REGION Network 2: 上行制动
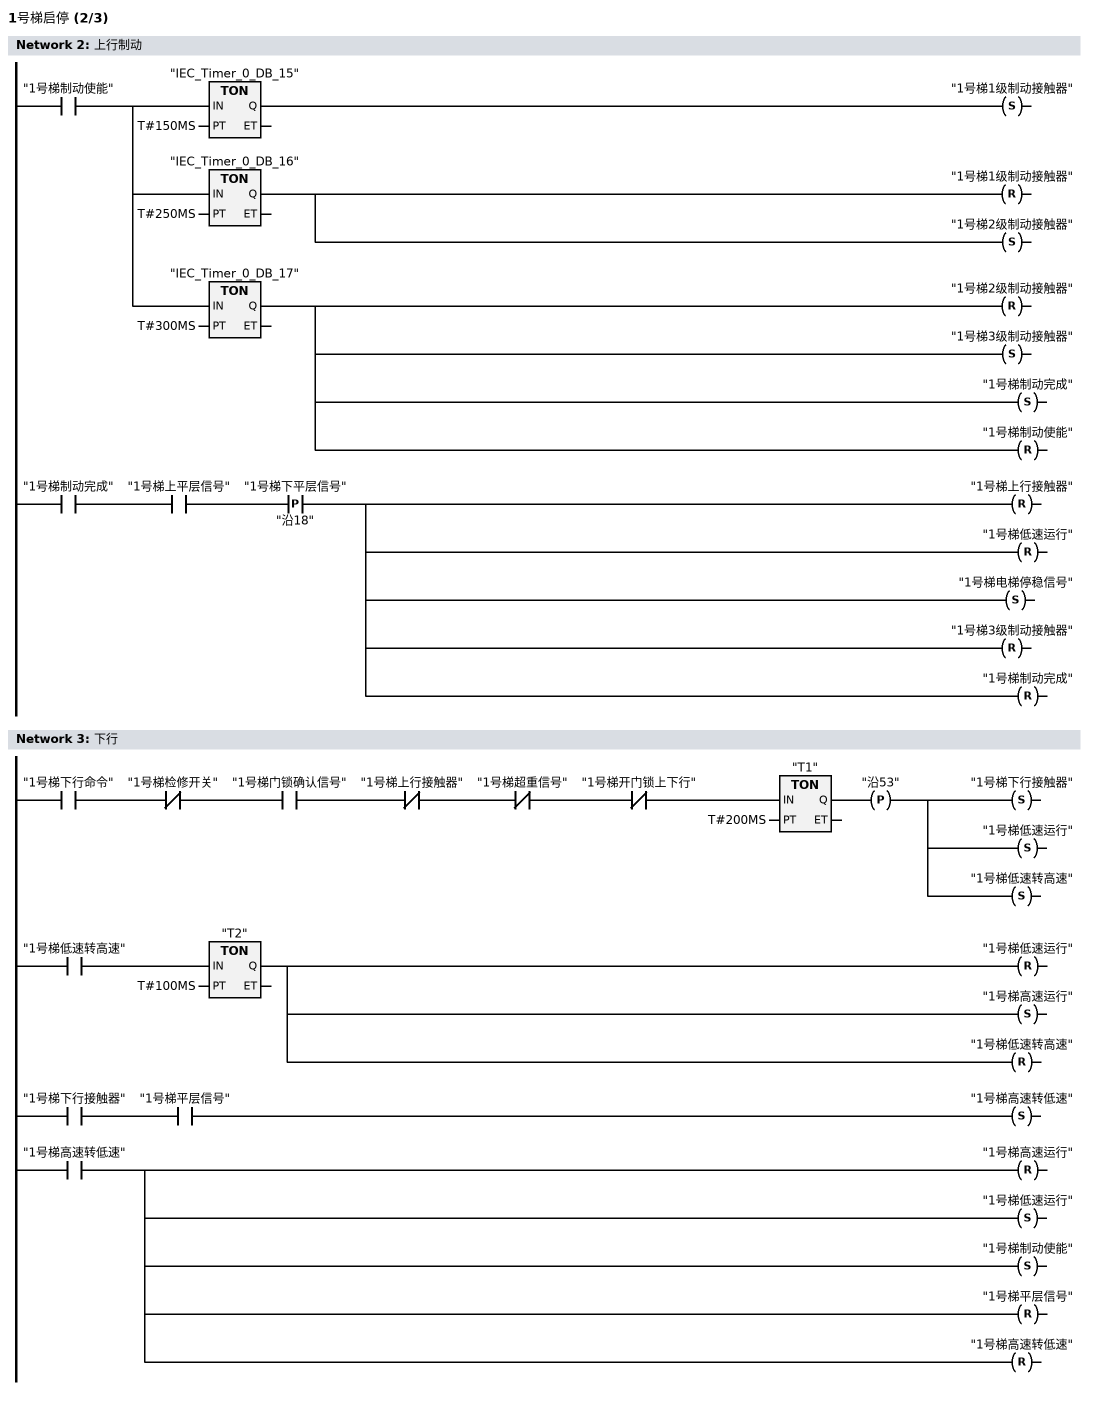
   "IEC_Timer_0_DB_15".TON(IN := "1号梯制动使能", PT := T#150MS);
   IF "IEC_Timer_0_DB_15".Q THEN "1号梯1级制动接触器" := TRUE; END_IF;
   "IEC_Timer_0_DB_16".TON(IN := "1号梯制动使能", PT := T#250MS);
   IF "IEC_Timer_0_DB_16".Q THEN
       "1号梯1级制动接触器" := FALSE;
       "1号梯2级制动接触器" := TRUE;
   END_IF;
   "IEC_Timer_0_DB_17".TON(IN := "1号梯制动使能", PT := T#300MS);
   IF "IEC_Timer_0_DB_17".Q THEN
       "1号梯2级制动接触器" := FALSE;
       "1号梯3级制动接触器" := TRUE;
       "1号梯制动完成" := TRUE;
       "1号梯制动使能" := FALSE;
   END_IF;
   #_w1 := "1号梯制动完成" AND "1号梯上平层信号" AND "1号梯下平层信号" AND NOT "沿18";   // rising edge of "1号梯下平层信号"
   "沿18" := "1号梯下平层信号";
   IF #_w1 THEN
       "1号梯上行接触器" := FALSE;
       "1号梯低速运行" := FALSE;
       "1号梯电梯停稳信号" := TRUE;
       "1号梯3级制动接触器" := FALSE;
       "1号梯制动完成" := FALSE;
   END_IF;
END_REGION

REGION Network 3: 下行
   "T1".TON(IN := "1号梯下行命令" AND NOT "1号梯检修开关" AND "1号梯门锁确认信号" AND NOT "1号梯上行接触器" AND NOT "1号梯超重信号" AND NOT "1号梯开门锁上下行",
            PT := T#200MS);
   #_w1 := "T1".Q AND NOT "沿53";   // rising edge
   "沿53" := "T1".Q;
   IF #_w1 THEN
       "1号梯下行接触器" := TRUE;
       "1号梯低速运行" := TRUE;
       "1号梯低速转高速" := TRUE;
   END_IF;
   "T2".TON(IN := "1号梯低速转高速", PT := T#100MS);
   IF "T2".Q THEN
       "1号梯低速运行" := FALSE;
       "1号梯高速运行" := TRUE;
       "1号梯低速转高速" := FALSE;
   END_IF;
   IF "1号梯下行接触器" AND "1号梯平层信号" THEN "1号梯高速转低速" := TRUE; END_IF;
   IF "1号梯高速转低速" THEN
       "1号梯高速运行" := FALSE;
       "1号梯低速运行" := TRUE;
       "1号梯制动使能" := TRUE;
       "1号梯平层信号" := FALSE;
       "1号梯高速转低速" := FALSE;
   END_IF;
END_REGION

REGION Network 4: 下行制动
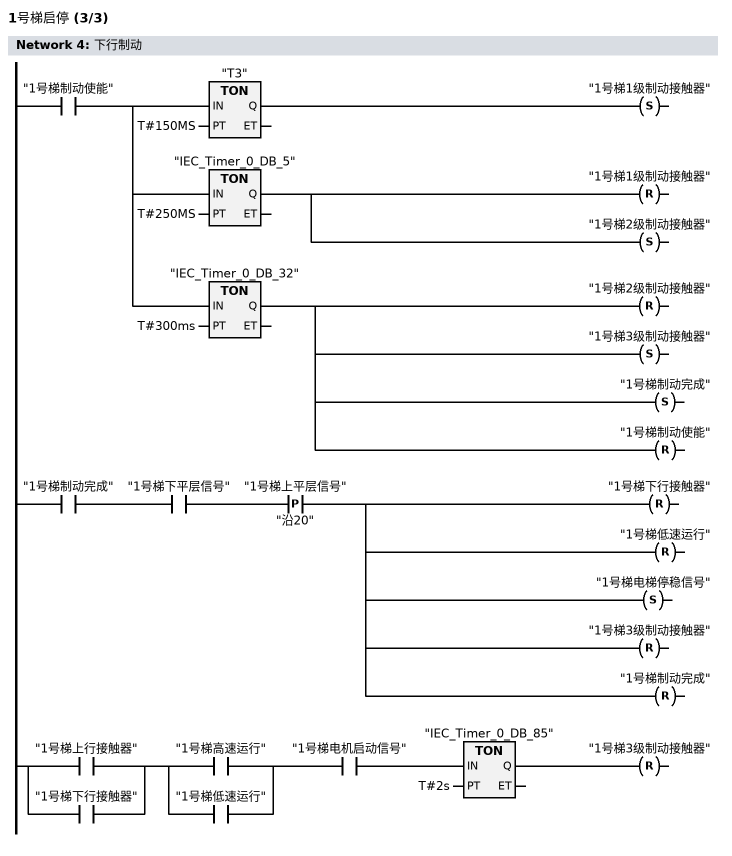
   "T3".TON(IN := "1号梯制动使能", PT := T#150MS);
   IF "T3".Q THEN "1号梯1级制动接触器" := TRUE; END_IF;
   "IEC_Timer_0_DB_5".TON(IN := "1号梯制动使能", PT := T#250MS);
   IF "IEC_Timer_0_DB_5".Q THEN
       "1号梯1级制动接触器" := FALSE;
       "1号梯2级制动接触器" := TRUE;
   END_IF;
   "IEC_Timer_0_DB_32".TON(IN := "1号梯制动使能", PT := T#300ms);
   IF "IEC_Timer_0_DB_32".Q THEN
       "1号梯2级制动接触器" := FALSE;
       "1号梯3级制动接触器" := TRUE;
       "1号梯制动完成" := TRUE;
       "1号梯制动使能" := FALSE;
   END_IF;
   #_w1 := "1号梯制动完成" AND "1号梯下平层信号" AND "1号梯上平层信号" AND NOT "沿20";   // rising edge of "1号梯上平层信号"
   "沿20" := "1号梯上平层信号";
   IF #_w1 THEN
       "1号梯下行接触器" := FALSE;
       "1号梯低速运行" := FALSE;
       "1号梯电梯停稳信号" := TRUE;
       "1号梯3级制动接触器" := FALSE;
       "1号梯制动完成" := FALSE;
   END_IF;
   "IEC_Timer_0_DB_85".TON(IN := ("1号梯上行接触器" OR "1号梯下行接触器") AND ("1号梯高速运行" OR "1号梯低速运行") AND "1号梯电机启动信号",
                           PT := T#2s);
   IF "IEC_Timer_0_DB_85".Q THEN "1号梯3级制动接触器" := FALSE; END_IF;
END_REGION
END_FUNCTION

FUNCTION "1号梯顺向截梯" : Void   // FC18, LAD
{ S7_Optimized_Access := 'TRUE' }
VERSION : 0.1
BEGIN

REGION Network 1: 上行拦截电梯
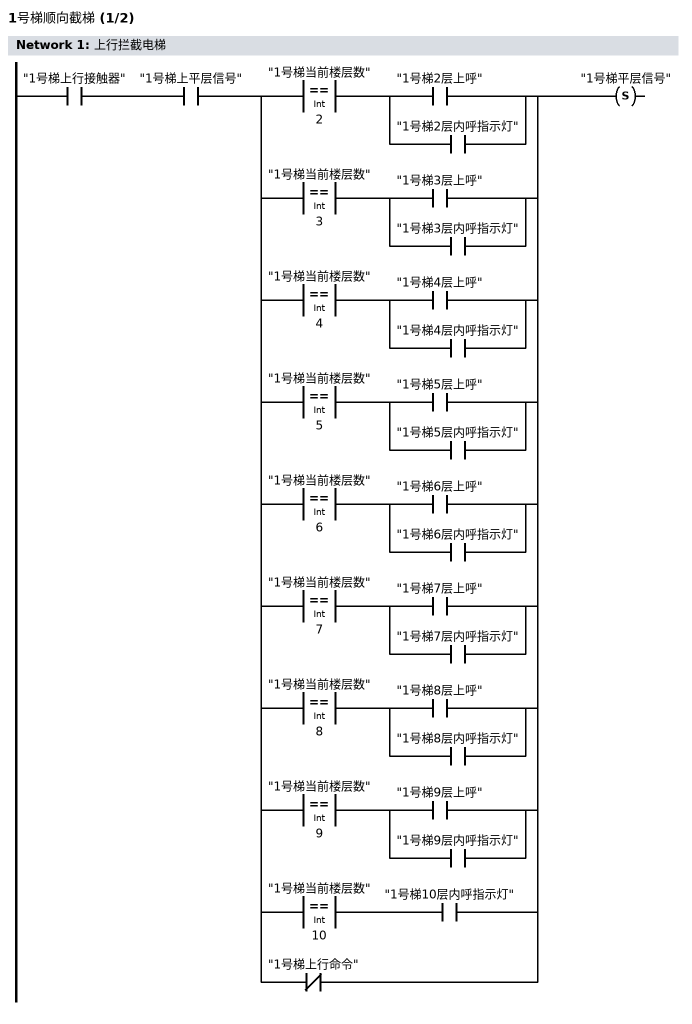
   RUNG wire#powerrail
      Contact( "1号梯上行接触器" )
      Contact( "1号梯上平层信号" )
      wire#w1
      { S7_Templates := "SrcType := Int" } EQ_Contact(in1 := "1号梯当前楼层数", in2 := 2)
      wire#w2
      Contact( "1号梯2层上呼" )
      wire#w3
      S_Coil( "1号梯平层信号" )
   END_RUNG
   RUNG wire#w2
      Contact( "1号梯2层内呼指示灯" )
   END_RUNG wire#w3
   RUNG wire#w1
      { S7_Templates := "SrcType := Int" } EQ_Contact(in1 := "1号梯当前楼层数", in2 := 3)
      wire#w4
      Contact( "1号梯3层上呼" )
   END_RUNG wire#w3
   RUNG wire#w4
      Contact( "1号梯3层内呼指示灯" )
   END_RUNG wire#w3
   RUNG wire#w1
      { S7_Templates := "SrcType := Int" } EQ_Contact(in1 := "1号梯当前楼层数", in2 := 4)
      wire#w5
      Contact( "1号梯4层上呼" )
   END_RUNG wire#w3
   RUNG wire#w5
      Contact( "1号梯4层内呼指示灯" )
   END_RUNG wire#w3
   RUNG wire#w1
      { S7_Templates := "SrcType := Int" } EQ_Contact(in1 := "1号梯当前楼层数", in2 := 5)
      wire#w6
      Contact( "1号梯5层上呼" )
   END_RUNG wire#w3
   RUNG wire#w6
      Contact( "1号梯5层内呼指示灯" )
   END_RUNG wire#w3
   RUNG wire#w1
      { S7_Templates := "SrcType := Int" } EQ_Contact(in1 := "1号梯当前楼层数", in2 := 6)
      wire#w7
      Contact( "1号梯6层上呼" )
   END_RUNG wire#w3
   RUNG wire#w7
      Contact( "1号梯6层内呼指示灯" )
   END_RUNG wire#w3
   RUNG wire#w1
      { S7_Templates := "SrcType := Int" } EQ_Contact(in1 := "1号梯当前楼层数", in2 := 7)
      wire#w8
      Contact( "1号梯7层上呼" )
   END_RUNG wire#w3
   RUNG wire#w8
      Contact( "1号梯7层内呼指示灯" )
   END_RUNG wire#w3
   RUNG wire#w1
      { S7_Templates := "SrcType := Int" } EQ_Contact(in1 := "1号梯当前楼层数", in2 := 8)
      wire#w9
      Contact( "1号梯8层上呼" )
   END_RUNG wire#w3
   RUNG wire#w9
      Contact( "1号梯8层内呼指示灯" )
   END_RUNG wire#w3
   RUNG wire#w1
      { S7_Templates := "SrcType := Int" } EQ_Contact(in1 := "1号梯当前楼层数", in2 := 9)
      wire#w10
      Contact( "1号梯9层上呼" )
   END_RUNG wire#w3
   RUNG wire#w10
      Contact( "1号梯9层内呼指示灯" )
   END_RUNG wire#w3
   RUNG wire#w1
      { S7_Templates := "SrcType := Int" } EQ_Contact(in1 := "1号梯当前楼层数", in2 := 10)
      Contact( "1号梯10层内呼指示灯" )
   END_RUNG wire#w3
   RUNG wire#w1
      I_Contact( "1号梯上行命令" )
   END_RUNG wire#w3
   // the same network as SCL:
   IF "1号梯上行接触器" AND "1号梯上平层信号" AND ((("1号梯当前楼层数" = 2) AND ("1号梯2层上呼" OR "1号梯2层内呼指示灯")) OR (("1号梯当前楼层数" = 3) AND ("1号梯3层上呼" OR "1号梯3层内呼指示灯")) OR (("1号梯当前楼层数" = 4) AND ("1号梯4层上呼" OR "1号梯4层内呼指示灯")) OR (("1号梯当前楼层数" = 5) AND ("1号梯5层上呼" OR "1号梯5层内呼指示灯")) OR (("1号梯当前楼层数" = 6) AND ("1号梯6层上呼" OR "1号梯6层内呼指示灯")) OR (("1号梯当前楼层数" = 7) AND ("1号梯7层上呼" OR "1号梯7层内呼指示灯")) OR (("1号梯当前楼层数" = 8) AND ("1号梯8层上呼" OR "1号梯8层内呼指示灯")) OR (("1号梯当前楼层数" = 9) AND ("1号梯9层上呼" OR "1号梯9层内呼指示灯")) OR (("1号梯当前楼层数" = 10) AND "1号梯10层内呼指示灯") OR NOT "1号梯上行命令") THEN
       "1号梯平层信号" := TRUE;
   END_IF;
END_REGION

REGION Network 2: 下行拦截电梯
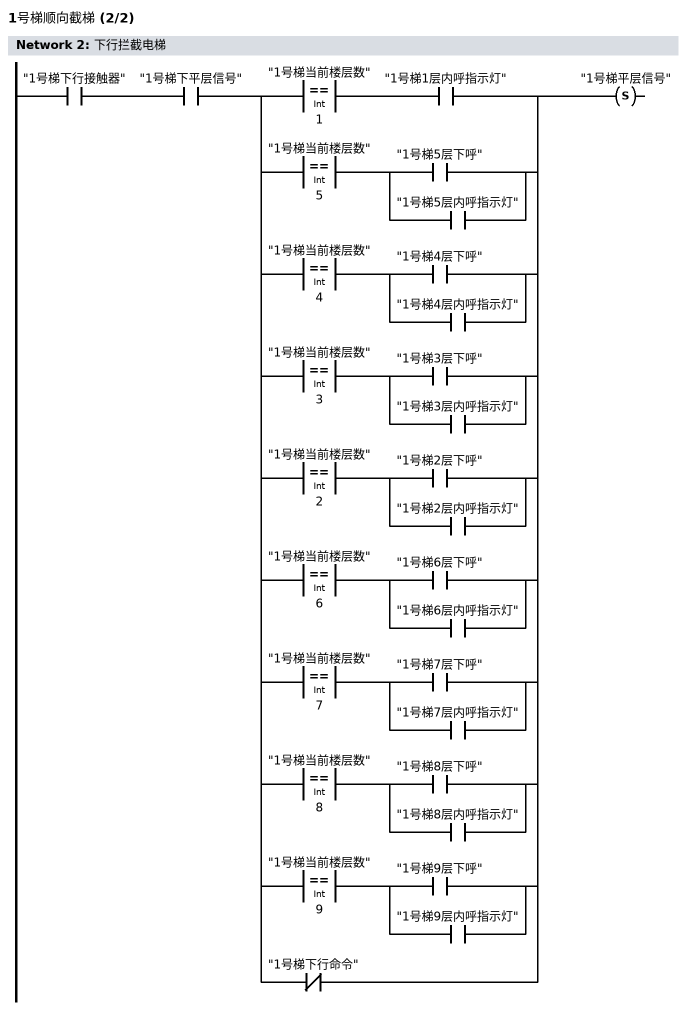
   RUNG wire#powerrail
      Contact( "1号梯下行接触器" )
      Contact( "1号梯下平层信号" )
      wire#w1
      { S7_Templates := "SrcType := Int" } EQ_Contact(in1 := "1号梯当前楼层数", in2 := 1)
      Contact( "1号梯1层内呼指示灯" )
      wire#w2
      S_Coil( "1号梯平层信号" )
   END_RUNG
   RUNG wire#w1
      { S7_Templates := "SrcType := Int" } EQ_Contact(in1 := "1号梯当前楼层数", in2 := 5)
      wire#w3
      Contact( "1号梯5层下呼" )
   END_RUNG wire#w2
   RUNG wire#w3
      Contact( "1号梯5层内呼指示灯" )
   END_RUNG wire#w2
   RUNG wire#w1
      { S7_Templates := "SrcType := Int" } EQ_Contact(in1 := "1号梯当前楼层数", in2 := 4)
      wire#w4
      Contact( "1号梯4层下呼" )
   END_RUNG wire#w2
   RUNG wire#w4
      Contact( "1号梯4层内呼指示灯" )
   END_RUNG wire#w2
   RUNG wire#w1
      { S7_Templates := "SrcType := Int" } EQ_Contact(in1 := "1号梯当前楼层数", in2 := 3)
      wire#w5
      Contact( "1号梯3层下呼" )
   END_RUNG wire#w2
   RUNG wire#w5
      Contact( "1号梯3层内呼指示灯" )
   END_RUNG wire#w2
   RUNG wire#w1
      { S7_Templates := "SrcType := Int" } EQ_Contact(in1 := "1号梯当前楼层数", in2 := 2)
      wire#w6
      Contact( "1号梯2层下呼" )
   END_RUNG wire#w2
   RUNG wire#w6
      Contact( "1号梯2层内呼指示灯" )
   END_RUNG wire#w2
   RUNG wire#w1
      { S7_Templates := "SrcType := Int" } EQ_Contact(in1 := "1号梯当前楼层数", in2 := 6)
      wire#w7
      Contact( "1号梯6层下呼" )
   END_RUNG wire#w2
   RUNG wire#w7
      Contact( "1号梯6层内呼指示灯" )
   END_RUNG wire#w2
   RUNG wire#w1
      { S7_Templates := "SrcType := Int" } EQ_Contact(in1 := "1号梯当前楼层数", in2 := 7)
      wire#w8
      Contact( "1号梯7层下呼" )
   END_RUNG wire#w2
   RUNG wire#w8
      Contact( "1号梯7层内呼指示灯" )
   END_RUNG wire#w2
   RUNG wire#w1
      { S7_Templates := "SrcType := Int" } EQ_Contact(in1 := "1号梯当前楼层数", in2 := 8)
      wire#w9
      Contact( "1号梯8层下呼" )
   END_RUNG wire#w2
   RUNG wire#w9
      Contact( "1号梯8层内呼指示灯" )
   END_RUNG wire#w2
   RUNG wire#w1
      { S7_Templates := "SrcType := Int" } EQ_Contact(in1 := "1号梯当前楼层数", in2 := 9)
      wire#w10
      Contact( "1号梯9层下呼" )
   END_RUNG wire#w2
   RUNG wire#w10
      Contact( "1号梯9层内呼指示灯" )
   END_RUNG wire#w2
   RUNG wire#w1
      I_Contact( "1号梯下行命令" )
   END_RUNG wire#w2
   // the same network as SCL:
   IF "1号梯下行接触器" AND "1号梯下平层信号" AND ((("1号梯当前楼层数" = 1) AND "1号梯1层内呼指示灯") OR (("1号梯当前楼层数" = 5) AND ("1号梯5层下呼" OR "1号梯5层内呼指示灯")) OR (("1号梯当前楼层数" = 4) AND ("1号梯4层下呼" OR "1号梯4层内呼指示灯")) OR (("1号梯当前楼层数" = 3) AND ("1号梯3层下呼" OR "1号梯3层内呼指示灯")) OR (("1号梯当前楼层数" = 2) AND ("1号梯2层下呼" OR "1号梯2层内呼指示灯")) OR (("1号梯当前楼层数" = 6) AND ("1号梯6层下呼" OR "1号梯6层内呼指示灯")) OR (("1号梯当前楼层数" = 7) AND ("1号梯7层下呼" OR "1号梯7层内呼指示灯")) OR (("1号梯当前楼层数" = 8) AND ("1号梯8层下呼" OR "1号梯8层内呼指示灯")) OR (("1号梯当前楼层数" = 9) AND ("1号梯9层下呼" OR "1号梯9层内呼指示灯")) OR NOT "1号梯下行命令") THEN
       "1号梯平层信号" := TRUE;
   END_IF;
END_REGION
END_FUNCTION

FUNCTION "1号梯轿内指示灯控制" : Void   // FC19, LAD
{ S7_Optimized_Access := 'TRUE' }
VERSION : 0.1
   VAR_TEMP   // added for the SCL form of the ladder/FBD networks
      _w1 : Bool;
      _w2 : Bool;
   END_VAR
BEGIN

REGION Network 1: 平层灭灯
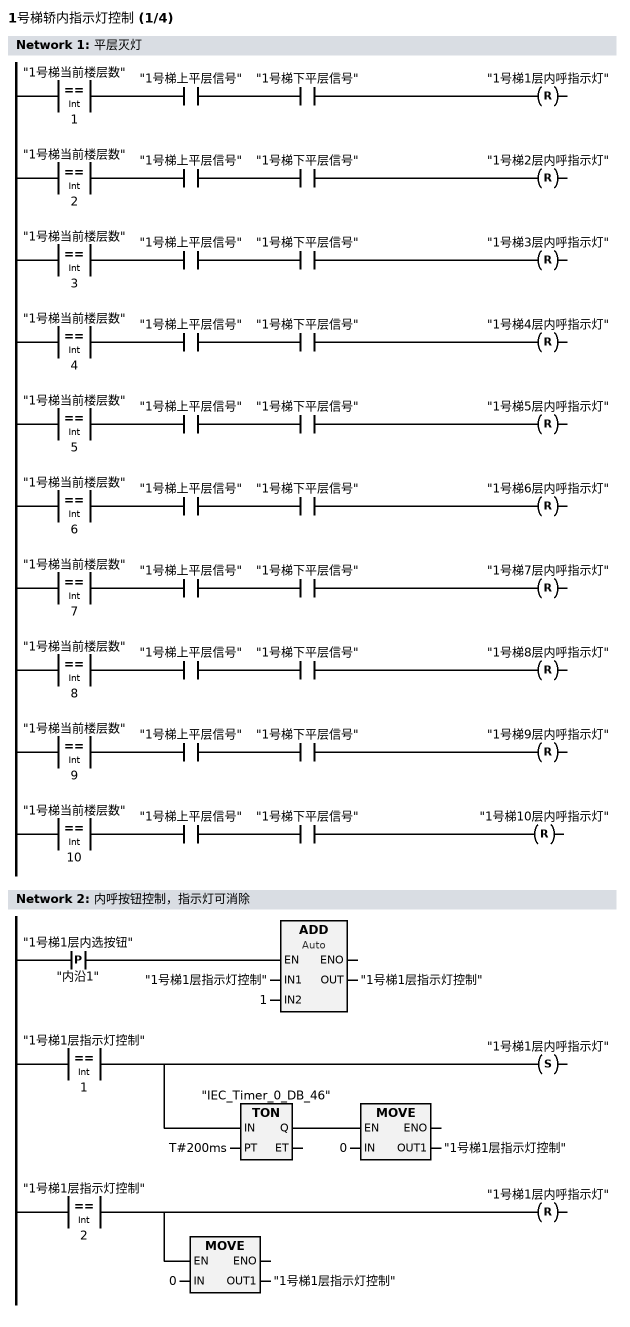
   RUNG wire#powerrail
      { S7_Templates := "SrcType := Int" } EQ_Contact(in1 := "1号梯当前楼层数", in2 := 1)
      Contact( "1号梯上平层信号" )
      Contact( "1号梯下平层信号" )
      R_Coil( "1号梯1层内呼指示灯" )
   END_RUNG
   RUNG wire#powerrail
      { S7_Templates := "SrcType := Int" } EQ_Contact(in1 := "1号梯当前楼层数", in2 := 2)
      Contact( "1号梯上平层信号" )
      Contact( "1号梯下平层信号" )
      R_Coil( "1号梯2层内呼指示灯" )
   END_RUNG
   RUNG wire#powerrail
      { S7_Templates := "SrcType := Int" } EQ_Contact(in1 := "1号梯当前楼层数", in2 := 3)
      Contact( "1号梯上平层信号" )
      Contact( "1号梯下平层信号" )
      R_Coil( "1号梯3层内呼指示灯" )
   END_RUNG
   RUNG wire#powerrail
      { S7_Templates := "SrcType := Int" } EQ_Contact(in1 := "1号梯当前楼层数", in2 := 4)
      Contact( "1号梯上平层信号" )
      Contact( "1号梯下平层信号" )
      R_Coil( "1号梯4层内呼指示灯" )
   END_RUNG
   RUNG wire#powerrail
      { S7_Templates := "SrcType := Int" } EQ_Contact(in1 := "1号梯当前楼层数", in2 := 5)
      Contact( "1号梯上平层信号" )
      Contact( "1号梯下平层信号" )
      R_Coil( "1号梯5层内呼指示灯" )
   END_RUNG
   RUNG wire#powerrail
      { S7_Templates := "SrcType := Int" } EQ_Contact(in1 := "1号梯当前楼层数", in2 := 6)
      Contact( "1号梯上平层信号" )
      Contact( "1号梯下平层信号" )
      R_Coil( "1号梯6层内呼指示灯" )
   END_RUNG
   RUNG wire#powerrail
      { S7_Templates := "SrcType := Int" } EQ_Contact(in1 := "1号梯当前楼层数", in2 := 7)
      Contact( "1号梯上平层信号" )
      Contact( "1号梯下平层信号" )
      R_Coil( "1号梯7层内呼指示灯" )
   END_RUNG
   RUNG wire#powerrail
      { S7_Templates := "SrcType := Int" } EQ_Contact(in1 := "1号梯当前楼层数", in2 := 8)
      Contact( "1号梯上平层信号" )
      Contact( "1号梯下平层信号" )
      R_Coil( "1号梯8层内呼指示灯" )
   END_RUNG
   RUNG wire#powerrail
      { S7_Templates := "SrcType := Int" } EQ_Contact(in1 := "1号梯当前楼层数", in2 := 9)
      Contact( "1号梯上平层信号" )
      Contact( "1号梯下平层信号" )
      R_Coil( "1号梯9层内呼指示灯" )
   END_RUNG
   RUNG wire#powerrail
      { S7_Templates := "SrcType := Int" } EQ_Contact(in1 := "1号梯当前楼层数", in2 := 10)
      Contact( "1号梯上平层信号" )
      Contact( "1号梯下平层信号" )
      R_Coil( "1号梯10层内呼指示灯" )
   END_RUNG
   // the same network as SCL:
   IF ("1号梯当前楼层数" = 1) AND "1号梯上平层信号" AND "1号梯下平层信号" THEN "1号梯1层内呼指示灯" := FALSE; END_IF;
   IF ("1号梯当前楼层数" = 2) AND "1号梯上平层信号" AND "1号梯下平层信号" THEN "1号梯2层内呼指示灯" := FALSE; END_IF;
   IF ("1号梯当前楼层数" = 3) AND "1号梯上平层信号" AND "1号梯下平层信号" THEN "1号梯3层内呼指示灯" := FALSE; END_IF;
   IF ("1号梯当前楼层数" = 4) AND "1号梯上平层信号" AND "1号梯下平层信号" THEN "1号梯4层内呼指示灯" := FALSE; END_IF;
   IF ("1号梯当前楼层数" = 5) AND "1号梯上平层信号" AND "1号梯下平层信号" THEN "1号梯5层内呼指示灯" := FALSE; END_IF;
   IF ("1号梯当前楼层数" = 6) AND "1号梯上平层信号" AND "1号梯下平层信号" THEN "1号梯6层内呼指示灯" := FALSE; END_IF;
   IF ("1号梯当前楼层数" = 7) AND "1号梯上平层信号" AND "1号梯下平层信号" THEN "1号梯7层内呼指示灯" := FALSE; END_IF;
   IF ("1号梯当前楼层数" = 8) AND "1号梯上平层信号" AND "1号梯下平层信号" THEN "1号梯8层内呼指示灯" := FALSE; END_IF;
   IF ("1号梯当前楼层数" = 9) AND "1号梯上平层信号" AND "1号梯下平层信号" THEN "1号梯9层内呼指示灯" := FALSE; END_IF;
   IF ("1号梯当前楼层数" = 10) AND "1号梯上平层信号" AND "1号梯下平层信号" THEN "1号梯10层内呼指示灯" := FALSE; END_IF;
END_REGION

REGION Network 2: 内呼按钮控制，指示灯可消除
   #_w1 := "1号梯1层内选按钮" AND NOT "内沿1";   // rising edge of "1号梯1层内选按钮"
   "内沿1" := "1号梯1层内选按钮";
   IF #_w1 THEN "1号梯1层指示灯控制" := "1号梯1层指示灯控制" + 1; END_IF;
   #_w2 := "1号梯1层指示灯控制" = 1;
   IF #_w2 THEN "1号梯1层内呼指示灯" := TRUE; END_IF;
   "IEC_Timer_0_DB_46".TON(IN := #_w2, PT := T#200ms);
   IF "IEC_Timer_0_DB_46".Q THEN "1号梯1层指示灯控制" := 0; END_IF;
   IF "1号梯1层指示灯控制" = 2 THEN
       "1号梯1层内呼指示灯" := FALSE;
       "1号梯1层指示灯控制" := 0;
   END_IF;
END_REGION

REGION Network 3: 内呼按钮控制，指示灯可消除
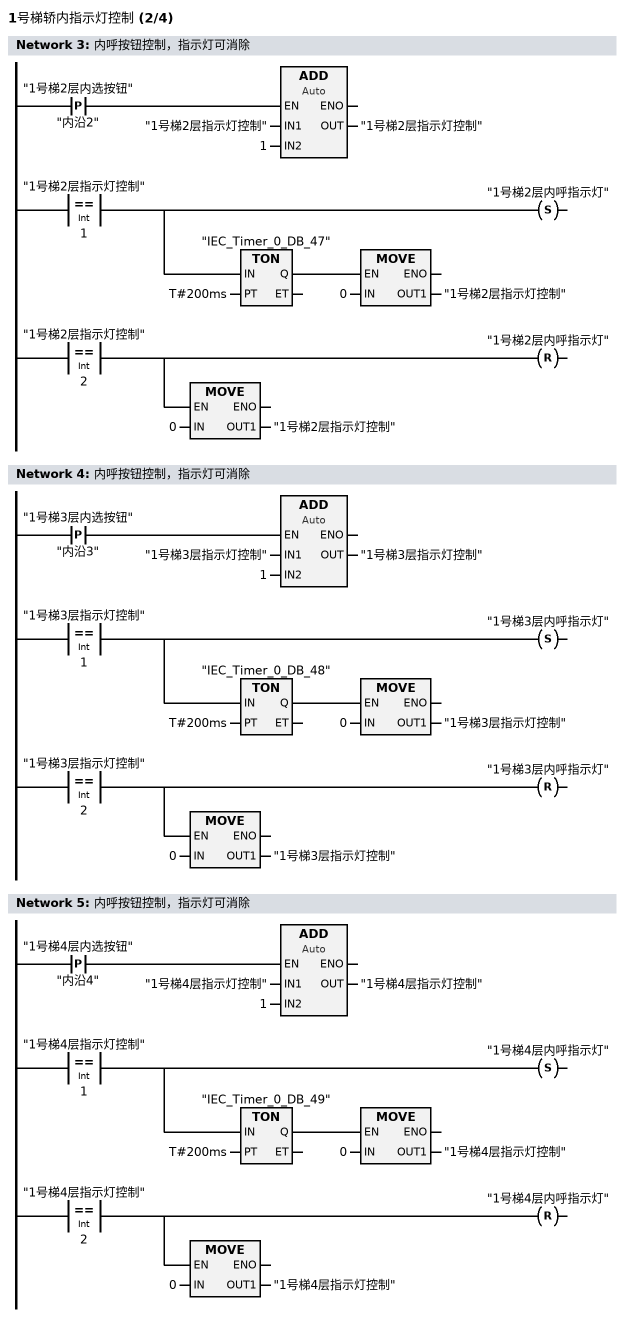
   #_w1 := "1号梯2层内选按钮" AND NOT "内沿2";   // rising edge of "1号梯2层内选按钮"
   "内沿2" := "1号梯2层内选按钮";
   IF #_w1 THEN "1号梯2层指示灯控制" := "1号梯2层指示灯控制" + 1; END_IF;
   #_w2 := "1号梯2层指示灯控制" = 1;
   IF #_w2 THEN "1号梯2层内呼指示灯" := TRUE; END_IF;
   "IEC_Timer_0_DB_47".TON(IN := #_w2, PT := T#200ms);
   IF "IEC_Timer_0_DB_47".Q THEN "1号梯2层指示灯控制" := 0; END_IF;
   IF "1号梯2层指示灯控制" = 2 THEN
       "1号梯2层内呼指示灯" := FALSE;
       "1号梯2层指示灯控制" := 0;
   END_IF;
END_REGION

REGION Network 4: 内呼按钮控制，指示灯可消除
   #_w1 := "1号梯3层内选按钮" AND NOT "内沿3";   // rising edge of "1号梯3层内选按钮"
   "内沿3" := "1号梯3层内选按钮";
   IF #_w1 THEN "1号梯3层指示灯控制" := "1号梯3层指示灯控制" + 1; END_IF;
   #_w2 := "1号梯3层指示灯控制" = 1;
   IF #_w2 THEN "1号梯3层内呼指示灯" := TRUE; END_IF;
   "IEC_Timer_0_DB_48".TON(IN := #_w2, PT := T#200ms);
   IF "IEC_Timer_0_DB_48".Q THEN "1号梯3层指示灯控制" := 0; END_IF;
   IF "1号梯3层指示灯控制" = 2 THEN
       "1号梯3层内呼指示灯" := FALSE;
       "1号梯3层指示灯控制" := 0;
   END_IF;
END_REGION

REGION Network 5: 内呼按钮控制，指示灯可消除
   #_w1 := "1号梯4层内选按钮" AND NOT "内沿4";   // rising edge of "1号梯4层内选按钮"
   "内沿4" := "1号梯4层内选按钮";
   IF #_w1 THEN "1号梯4层指示灯控制" := "1号梯4层指示灯控制" + 1; END_IF;
   #_w2 := "1号梯4层指示灯控制" = 1;
   IF #_w2 THEN "1号梯4层内呼指示灯" := TRUE; END_IF;
   "IEC_Timer_0_DB_49".TON(IN := #_w2, PT := T#200ms);
   IF "IEC_Timer_0_DB_49".Q THEN "1号梯4层指示灯控制" := 0; END_IF;
   IF "1号梯4层指示灯控制" = 2 THEN
       "1号梯4层内呼指示灯" := FALSE;
       "1号梯4层指示灯控制" := 0;
   END_IF;
END_REGION

REGION Network 6: 内呼按钮控制，指示灯可消除
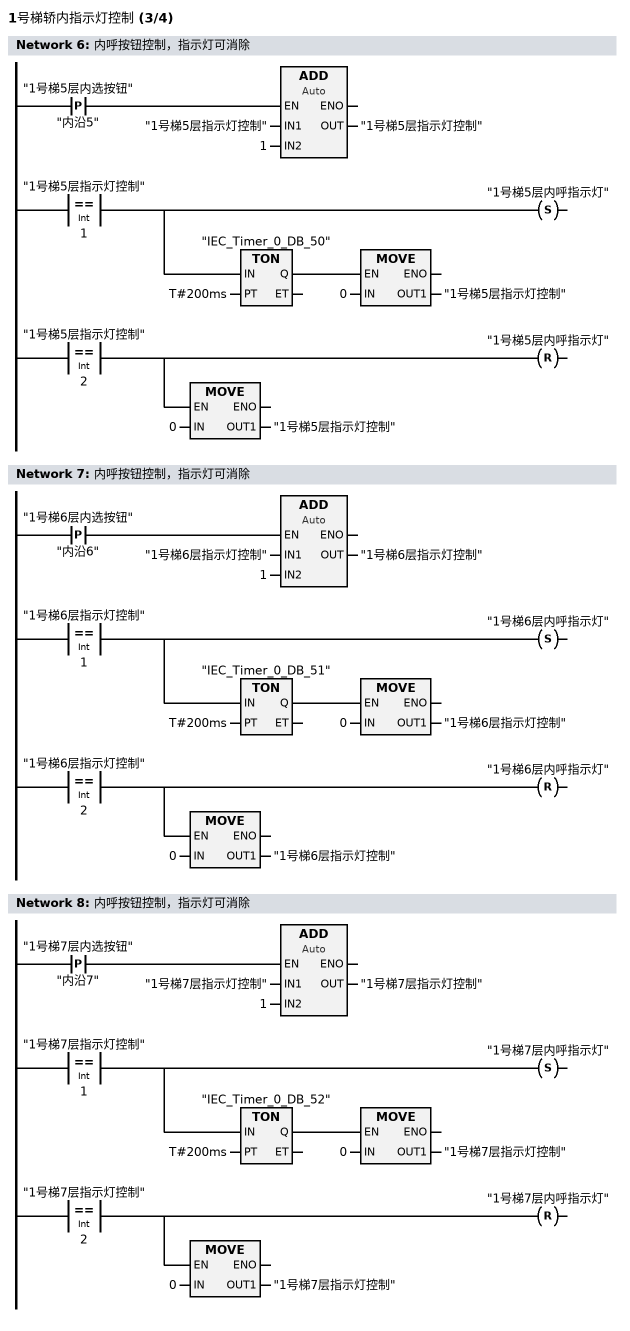
   #_w1 := "1号梯5层内选按钮" AND NOT "内沿5";   // rising edge of "1号梯5层内选按钮"
   "内沿5" := "1号梯5层内选按钮";
   IF #_w1 THEN "1号梯5层指示灯控制" := "1号梯5层指示灯控制" + 1; END_IF;
   #_w2 := "1号梯5层指示灯控制" = 1;
   IF #_w2 THEN "1号梯5层内呼指示灯" := TRUE; END_IF;
   "IEC_Timer_0_DB_50".TON(IN := #_w2, PT := T#200ms);
   IF "IEC_Timer_0_DB_50".Q THEN "1号梯5层指示灯控制" := 0; END_IF;
   IF "1号梯5层指示灯控制" = 2 THEN
       "1号梯5层内呼指示灯" := FALSE;
       "1号梯5层指示灯控制" := 0;
   END_IF;
END_REGION

REGION Network 7: 内呼按钮控制，指示灯可消除
   #_w1 := "1号梯6层内选按钮" AND NOT "内沿6";   // rising edge of "1号梯6层内选按钮"
   "内沿6" := "1号梯6层内选按钮";
   IF #_w1 THEN "1号梯6层指示灯控制" := "1号梯6层指示灯控制" + 1; END_IF;
   #_w2 := "1号梯6层指示灯控制" = 1;
   IF #_w2 THEN "1号梯6层内呼指示灯" := TRUE; END_IF;
   "IEC_Timer_0_DB_51".TON(IN := #_w2, PT := T#200ms);
   IF "IEC_Timer_0_DB_51".Q THEN "1号梯6层指示灯控制" := 0; END_IF;
   IF "1号梯6层指示灯控制" = 2 THEN
       "1号梯6层内呼指示灯" := FALSE;
       "1号梯6层指示灯控制" := 0;
   END_IF;
END_REGION

REGION Network 8: 内呼按钮控制，指示灯可消除
   #_w1 := "1号梯7层内选按钮" AND NOT "内沿7";   // rising edge of "1号梯7层内选按钮"
   "内沿7" := "1号梯7层内选按钮";
   IF #_w1 THEN "1号梯7层指示灯控制" := "1号梯7层指示灯控制" + 1; END_IF;
   #_w2 := "1号梯7层指示灯控制" = 1;
   IF #_w2 THEN "1号梯7层内呼指示灯" := TRUE; END_IF;
   "IEC_Timer_0_DB_52".TON(IN := #_w2, PT := T#200ms);
   IF "IEC_Timer_0_DB_52".Q THEN "1号梯7层指示灯控制" := 0; END_IF;
   IF "1号梯7层指示灯控制" = 2 THEN
       "1号梯7层内呼指示灯" := FALSE;
       "1号梯7层指示灯控制" := 0;
   END_IF;
END_REGION

REGION Network 9: 内呼按钮控制，指示灯可消除
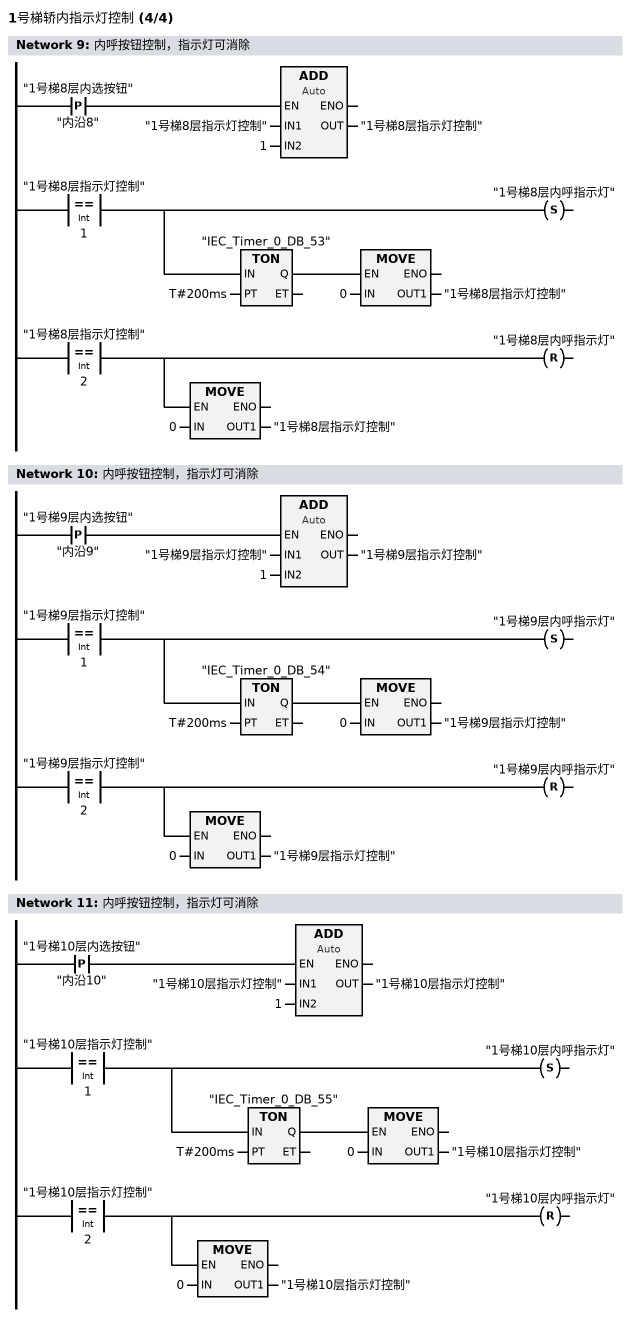
   #_w1 := "1号梯8层内选按钮" AND NOT "内沿8";   // rising edge of "1号梯8层内选按钮"
   "内沿8" := "1号梯8层内选按钮";
   IF #_w1 THEN "1号梯8层指示灯控制" := "1号梯8层指示灯控制" + 1; END_IF;
   #_w2 := "1号梯8层指示灯控制" = 1;
   IF #_w2 THEN "1号梯8层内呼指示灯" := TRUE; END_IF;
   "IEC_Timer_0_DB_53".TON(IN := #_w2, PT := T#200ms);
   IF "IEC_Timer_0_DB_53".Q THEN "1号梯8层指示灯控制" := 0; END_IF;
   IF "1号梯8层指示灯控制" = 2 THEN
       "1号梯8层内呼指示灯" := FALSE;
       "1号梯8层指示灯控制" := 0;
   END_IF;
END_REGION

REGION Network 10: 内呼按钮控制，指示灯可消除
   #_w1 := "1号梯9层内选按钮" AND NOT "内沿9";   // rising edge of "1号梯9层内选按钮"
   "内沿9" := "1号梯9层内选按钮";
   IF #_w1 THEN "1号梯9层指示灯控制" := "1号梯9层指示灯控制" + 1; END_IF;
   #_w2 := "1号梯9层指示灯控制" = 1;
   IF #_w2 THEN "1号梯9层内呼指示灯" := TRUE; END_IF;
   "IEC_Timer_0_DB_54".TON(IN := #_w2, PT := T#200ms);
   IF "IEC_Timer_0_DB_54".Q THEN "1号梯9层指示灯控制" := 0; END_IF;
   IF "1号梯9层指示灯控制" = 2 THEN
       "1号梯9层内呼指示灯" := FALSE;
       "1号梯9层指示灯控制" := 0;
   END_IF;
END_REGION

REGION Network 11: 内呼按钮控制，指示灯可消除
   #_w1 := "1号梯10层内选按钮" AND NOT "内沿10";   // rising edge of "1号梯10层内选按钮"
   "内沿10" := "1号梯10层内选按钮";
   IF #_w1 THEN "1号梯10层指示灯控制" := "1号梯10层指示灯控制" + 1; END_IF;
   #_w2 := "1号梯10层指示灯控制" = 1;
   IF #_w2 THEN "1号梯10层内呼指示灯" := TRUE; END_IF;
   "IEC_Timer_0_DB_55".TON(IN := #_w2, PT := T#200ms);
   IF "IEC_Timer_0_DB_55".Q THEN "1号梯10层指示灯控制" := 0; END_IF;
   IF "1号梯10层指示灯控制" = 2 THEN
       "1号梯10层内呼指示灯" := FALSE;
       "1号梯10层指示灯控制" := 0;
   END_IF;
END_REGION
END_FUNCTION

FUNCTION "1号梯保护程序" : Void   // FC20, LAD
{ S7_Optimized_Access := 'TRUE' }
VERSION : 0.1
BEGIN

REGION Network 1: 休眠管理
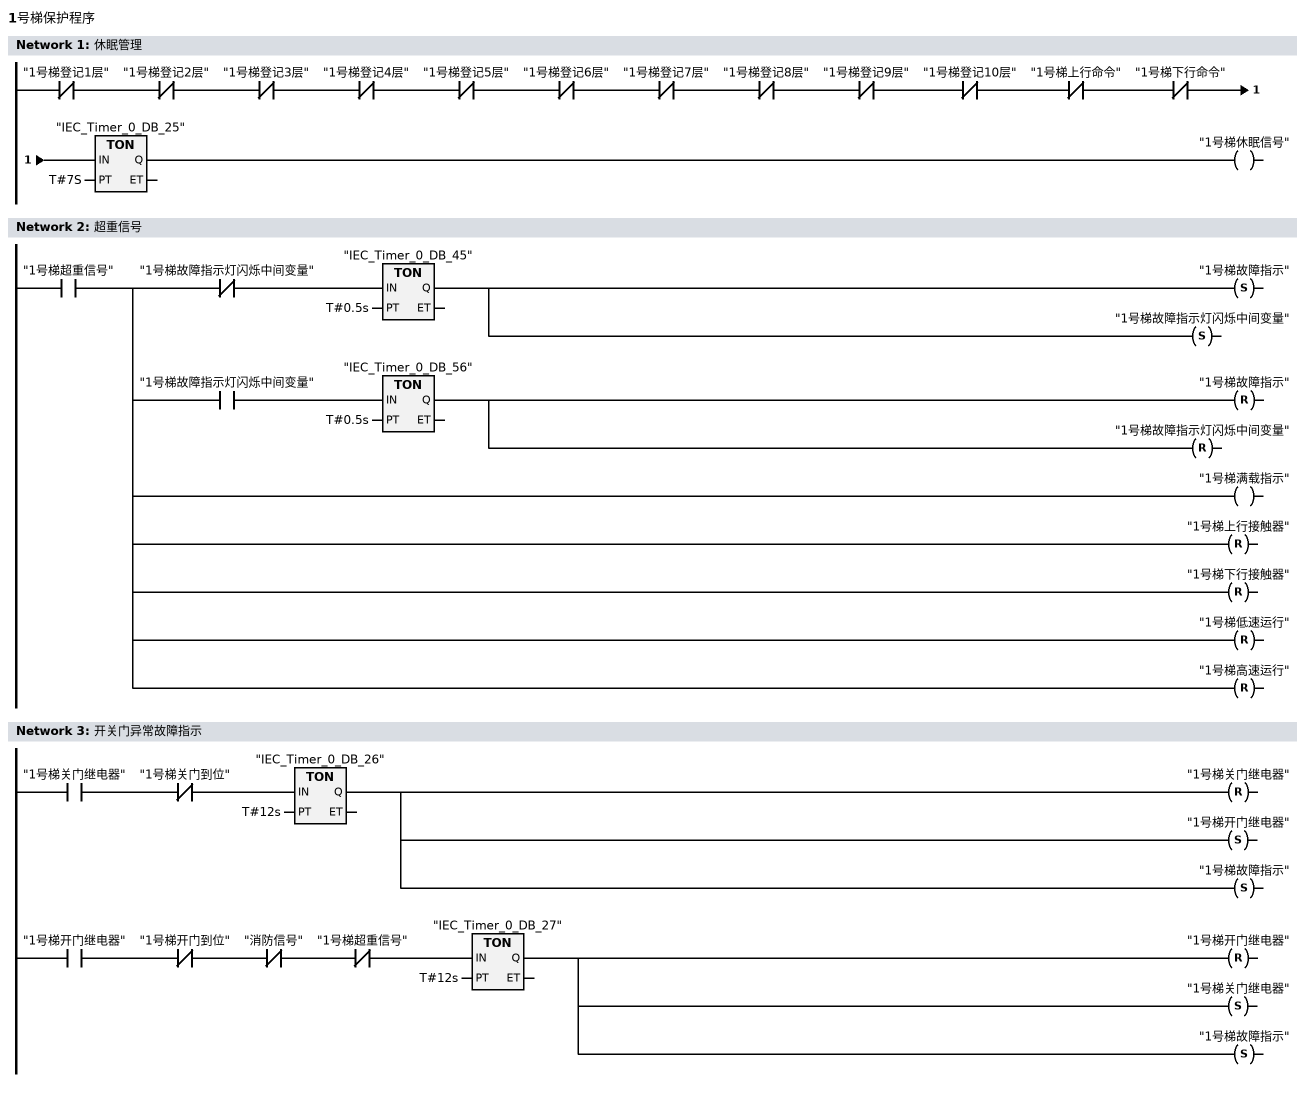
   "IEC_Timer_0_DB_25".TON(IN := NOT "1号梯登记1层" AND NOT "1号梯登记2层" AND NOT "1号梯登记3层" AND NOT "1号梯登记4层" AND NOT "1号梯登记5层" AND NOT "1号梯登记6层" AND NOT "1号梯登记7层" AND NOT "1号梯登记8层" AND NOT "1号梯登记9层" AND NOT "1号梯登记10层" AND NOT "1号梯上行命令" AND NOT "1号梯下行命令",
                           PT := T#7S);
   "1号梯休眠信号" := "IEC_Timer_0_DB_25".Q;
END_REGION

REGION Network 2: 超重信号
   "IEC_Timer_0_DB_45".TON(IN := "1号梯超重信号" AND NOT "1号梯故障指示灯闪烁中间变量", PT := T#0.5s);
   IF "IEC_Timer_0_DB_45".Q THEN
       "1号梯故障指示" := TRUE;
       "1号梯故障指示灯闪烁中间变量" := TRUE;
   END_IF;
   "IEC_Timer_0_DB_56".TON(IN := "1号梯超重信号" AND "1号梯故障指示灯闪烁中间变量", PT := T#0.5s);
   IF "IEC_Timer_0_DB_56".Q THEN
       "1号梯故障指示" := FALSE;
       "1号梯故障指示灯闪烁中间变量" := FALSE;
   END_IF;
   "1号梯满载指示" := "1号梯超重信号";
   IF "1号梯超重信号" THEN
       "1号梯上行接触器" := FALSE;
       "1号梯下行接触器" := FALSE;
       "1号梯低速运行" := FALSE;
       "1号梯高速运行" := FALSE;
   END_IF;
END_REGION

REGION Network 3: 开关门异常故障指示
   "IEC_Timer_0_DB_26".TON(IN := "1号梯关门继电器" AND NOT "1号梯关门到位", PT := T#12s);
   IF "IEC_Timer_0_DB_26".Q THEN
       "1号梯关门继电器" := FALSE;
       "1号梯开门继电器" := TRUE;
       "1号梯故障指示" := TRUE;
   END_IF;
   "IEC_Timer_0_DB_27".TON(IN := "1号梯开门继电器" AND NOT "1号梯开门到位" AND NOT "消防信号" AND NOT "1号梯超重信号", PT := T#12s);
   IF "IEC_Timer_0_DB_27".Q THEN
       "1号梯开门继电器" := FALSE;
       "1号梯关门继电器" := TRUE;
       "1号梯故障指示" := TRUE;
   END_IF;
END_REGION
END_FUNCTION

FUNCTION "1号梯错误指令消除" : Void   // FC21, LAD
{ S7_Optimized_Access := 'TRUE' }
VERSION : 0.1
BEGIN

REGION Network 1: 最上端/最下端时， 消除内呼信号
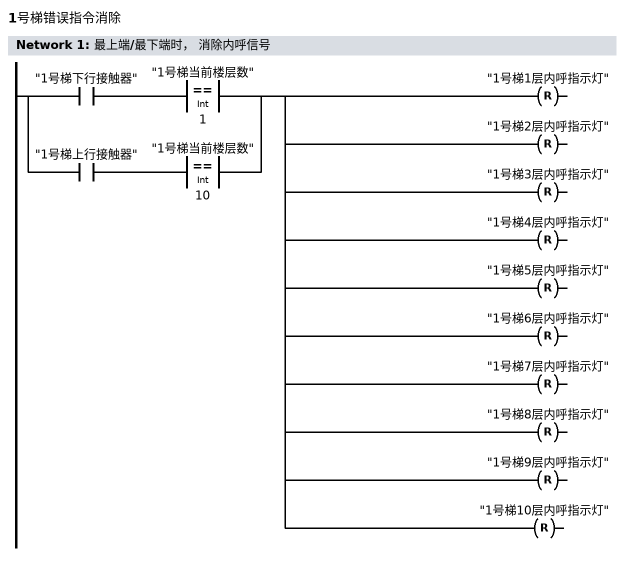
   RUNG wire#powerrail
      Contact( "1号梯下行接触器" )
      { S7_Templates := "SrcType := Int" } EQ_Contact(in1 := "1号梯当前楼层数", in2 := 1)
      wire#w1
      R_Coil( "1号梯1层内呼指示灯" )
   END_RUNG
   RUNG wire#powerrail
      Contact( "1号梯上行接触器" )
      { S7_Templates := "SrcType := Int" } EQ_Contact(in1 := "1号梯当前楼层数", in2 := 10)
   END_RUNG wire#w1
   RUNG wire#w1
      R_Coil( "1号梯2层内呼指示灯" )
   END_RUNG
   RUNG wire#w1
      R_Coil( "1号梯3层内呼指示灯" )
   END_RUNG
   RUNG wire#w1
      R_Coil( "1号梯4层内呼指示灯" )
   END_RUNG
   RUNG wire#w1
      R_Coil( "1号梯5层内呼指示灯" )
   END_RUNG
   RUNG wire#w1
      R_Coil( "1号梯6层内呼指示灯" )
   END_RUNG
   RUNG wire#w1
      R_Coil( "1号梯7层内呼指示灯" )
   END_RUNG
   RUNG wire#w1
      R_Coil( "1号梯8层内呼指示灯" )
   END_RUNG
   RUNG wire#w1
      R_Coil( "1号梯9层内呼指示灯" )
   END_RUNG
   RUNG wire#w1
      R_Coil( "1号梯10层内呼指示灯" )
   END_RUNG
   // the same network as SCL:
   IF ("1号梯下行接触器" AND ("1号梯当前楼层数" = 1)) OR ("1号梯上行接触器" AND ("1号梯当前楼层数" = 10)) THEN
       "1号梯1层内呼指示灯" := FALSE;
       "1号梯2层内呼指示灯" := FALSE;
       "1号梯3层内呼指示灯" := FALSE;
       "1号梯4层内呼指示灯" := FALSE;
       "1号梯5层内呼指示灯" := FALSE;
       "1号梯6层内呼指示灯" := FALSE;
       "1号梯7层内呼指示灯" := FALSE;
       "1号梯8层内呼指示灯" := FALSE;
       "1号梯9层内呼指示灯" := FALSE;
       "1号梯10层内呼指示灯" := FALSE;
   END_IF;
END_REGION
END_FUNCTION

FUNCTION "1号梯检修" : Void   // FC22, LAD
{ S7_Optimized_Access := 'TRUE' }
VERSION : 0.1
   VAR_TEMP   // added for the SCL form of the ladder/FBD networks
      _w1 : Bool;
   END_VAR
BEGIN

REGION Network 1: 检修
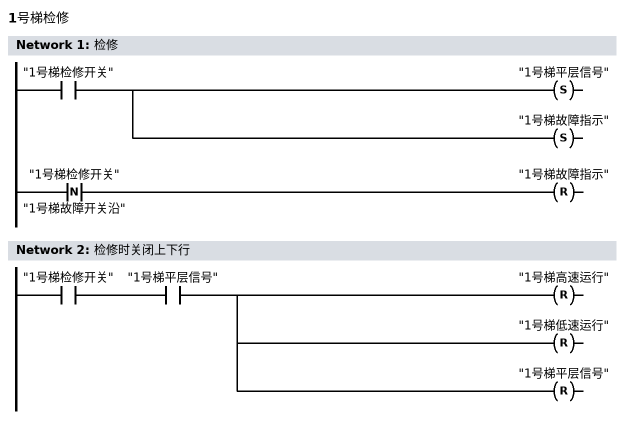
   RUNG wire#powerrail
      Contact( "1号梯检修开关" )
      wire#w1
      S_Coil( "1号梯平层信号" )
   END_RUNG
   RUNG wire#w1
      S_Coil( "1号梯故障指示" )
   END_RUNG
   RUNG wire#powerrail
      N_Contact(operand := "1号梯检修开关", bit := "1号梯故障开关沿")
      R_Coil( "1号梯故障指示" )
   END_RUNG
   // the same network as SCL:
   IF "1号梯检修开关" THEN
       "1号梯平层信号" := TRUE;
       "1号梯故障指示" := TRUE;
   END_IF;
   #_w1 := NOT "1号梯检修开关" AND "1号梯故障开关沿";   // falling edge of "1号梯检修开关"
   "1号梯故障开关沿" := "1号梯检修开关";
   IF #_w1 THEN "1号梯故障指示" := FALSE; END_IF;
END_REGION

REGION Network 2: 检修时关闭上下行
   RUNG wire#powerrail
      Contact( "1号梯检修开关" )
      Contact( "1号梯平层信号" )
      wire#w1
      R_Coil( "1号梯高速运行" )
   END_RUNG
   RUNG wire#w1
      R_Coil( "1号梯低速运行" )
   END_RUNG
   RUNG wire#w1
      R_Coil( "1号梯平层信号" )
   END_RUNG
   // the same network as SCL:
   IF "1号梯检修开关" AND "1号梯平层信号" THEN
       "1号梯高速运行" := FALSE;
       "1号梯低速运行" := FALSE;
       "1号梯平层信号" := FALSE;
   END_IF;
END_REGION
END_FUNCTION

FUNCTION "3号梯数码管显示" : Void   // FC23, LAD
{ S7_Optimized_Access := 'TRUE' }
VERSION : 0.1
   VAR_TEMP   // added for the SCL form of the ladder/FBD networks
      _w1 : Bool;
      _w2 : Bool;
      _w3 : Bool;
      _w4 : Bool;
      _w5 : Bool;
      _w6 : Bool;
      _w7 : Bool;
      _w8 : Bool;
      _w9 : Bool;
      _w10 : Bool;
      _w11 : Bool;
      _w12 : Bool;
      _w13 : Bool;
      _w14 : Bool;
      _w15 : Bool;
      _w16 : Bool;
      _w17 : Bool;
      _w18 : Bool;
      _w19 : Bool;
      _w20 : Bool;
   END_VAR
BEGIN

REGION Network 1: 根据楼层显示数码管
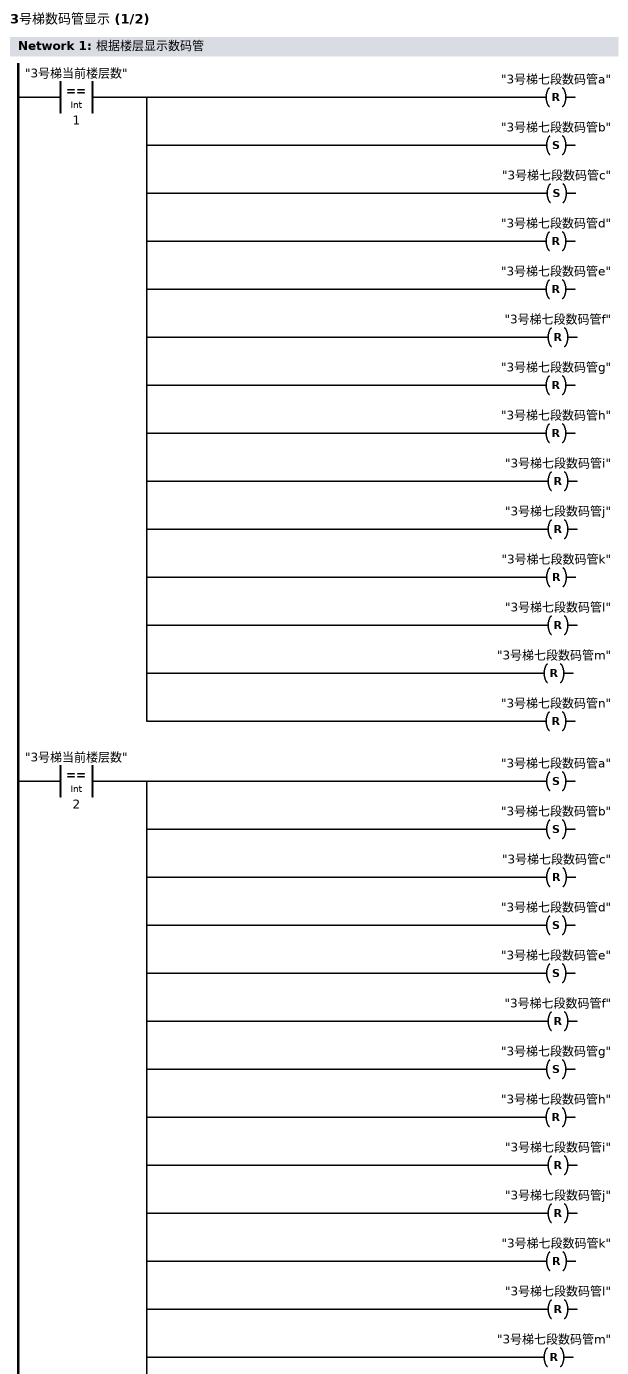
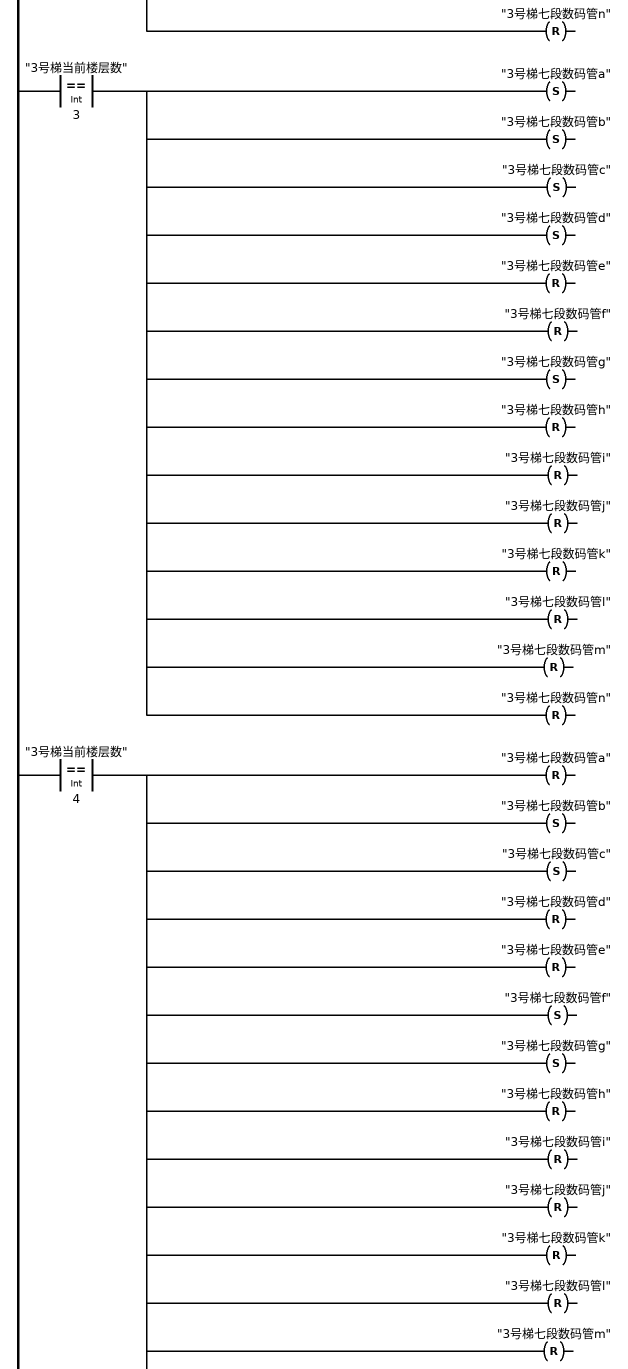
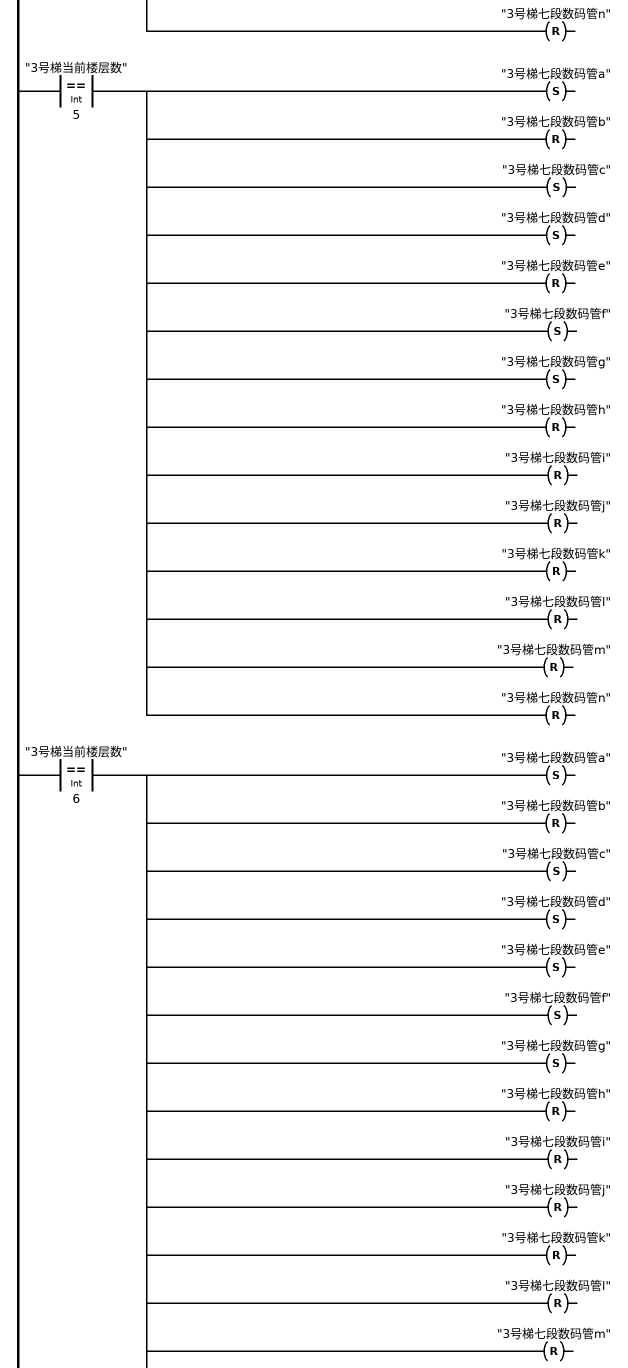
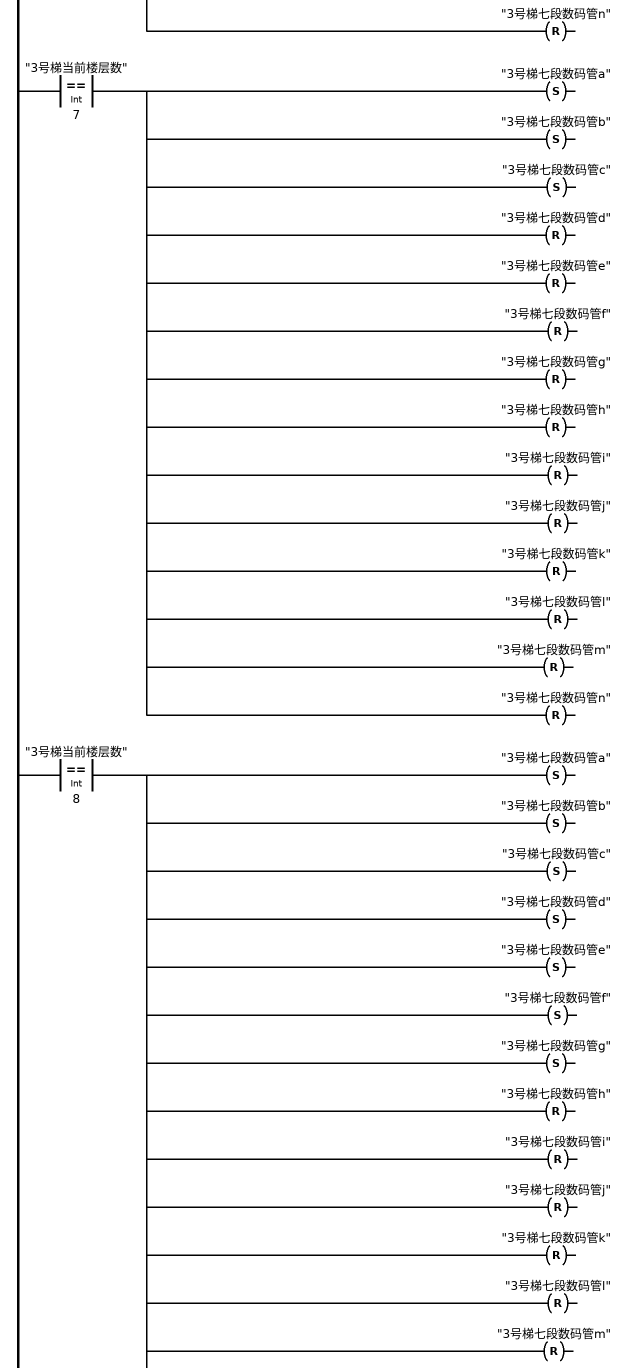
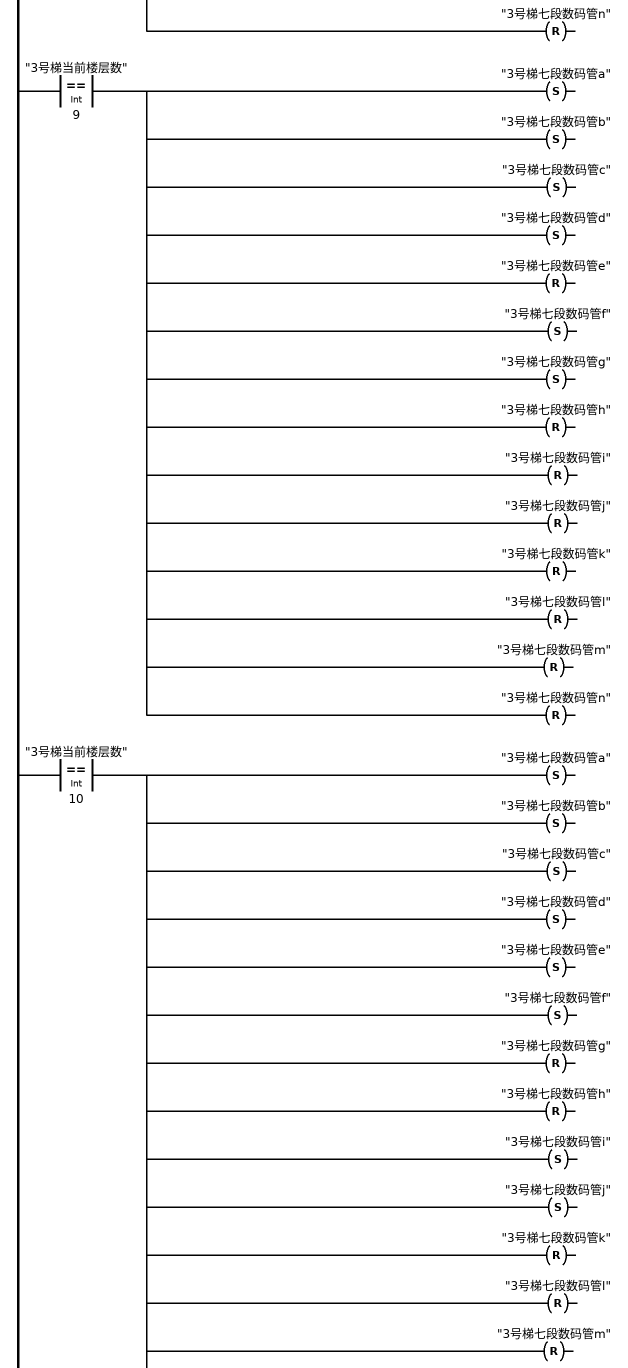
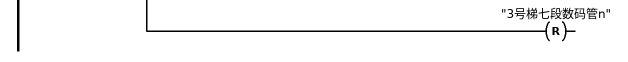
   RUNG wire#powerrail
      { S7_Templates := "SrcType := Int" } EQ_Contact(in1 := "3号梯当前楼层数", in2 := 1)
      wire#w1
      R_Coil( "3号梯七段数码管a" )
   END_RUNG
   RUNG wire#w1
      S_Coil( "3号梯七段数码管b" )
   END_RUNG
   RUNG wire#w1
      S_Coil( "3号梯七段数码管c" )
   END_RUNG
   RUNG wire#w1
      R_Coil( "3号梯七段数码管d" )
   END_RUNG
   RUNG wire#w1
      R_Coil( "3号梯七段数码管e" )
   END_RUNG
   RUNG wire#w1
      R_Coil( "3号梯七段数码管f" )
   END_RUNG
   RUNG wire#w1
      R_Coil( "3号梯七段数码管g" )
   END_RUNG
   RUNG wire#w1
      R_Coil( "3号梯七段数码管h" )
   END_RUNG
   RUNG wire#w1
      R_Coil( "3号梯七段数码管i" )
   END_RUNG
   RUNG wire#w1
      R_Coil( "3号梯七段数码管j" )
   END_RUNG
   RUNG wire#w1
      R_Coil( "3号梯七段数码管k" )
   END_RUNG
   RUNG wire#w1
      R_Coil( "3号梯七段数码管l" )
   END_RUNG
   RUNG wire#w1
      R_Coil( "3号梯七段数码管m" )
   END_RUNG
   RUNG wire#w1
      R_Coil( "3号梯七段数码管n" )
   END_RUNG
   RUNG wire#powerrail
      { S7_Templates := "SrcType := Int" } EQ_Contact(in1 := "3号梯当前楼层数", in2 := 2)
      wire#w2
      S_Coil( "3号梯七段数码管a" )
   END_RUNG
   RUNG wire#w2
      S_Coil( "3号梯七段数码管b" )
   END_RUNG
   RUNG wire#w2
      R_Coil( "3号梯七段数码管c" )
   END_RUNG
   RUNG wire#w2
      S_Coil( "3号梯七段数码管d" )
   END_RUNG
   RUNG wire#w2
      S_Coil( "3号梯七段数码管e" )
   END_RUNG
   RUNG wire#w2
      R_Coil( "3号梯七段数码管f" )
   END_RUNG
   RUNG wire#w2
      S_Coil( "3号梯七段数码管g" )
   END_RUNG
   RUNG wire#w2
      R_Coil( "3号梯七段数码管h" )
   END_RUNG
   RUNG wire#w2
      R_Coil( "3号梯七段数码管i" )
   END_RUNG
   RUNG wire#w2
      R_Coil( "3号梯七段数码管j" )
   END_RUNG
   RUNG wire#w2
      R_Coil( "3号梯七段数码管k" )
   END_RUNG
   RUNG wire#w2
      R_Coil( "3号梯七段数码管l" )
   END_RUNG
   RUNG wire#w2
      R_Coil( "3号梯七段数码管m" )
   END_RUNG
   RUNG wire#w2
      R_Coil( "3号梯七段数码管n" )
   END_RUNG
   RUNG wire#powerrail
      { S7_Templates := "SrcType := Int" } EQ_Contact(in1 := "3号梯当前楼层数", in2 := 3)
      wire#w3
      S_Coil( "3号梯七段数码管a" )
   END_RUNG
   RUNG wire#w3
      S_Coil( "3号梯七段数码管b" )
   END_RUNG
   RUNG wire#w3
      S_Coil( "3号梯七段数码管c" )
   END_RUNG
   RUNG wire#w3
      S_Coil( "3号梯七段数码管d" )
   END_RUNG
   RUNG wire#w3
      R_Coil( "3号梯七段数码管e" )
   END_RUNG
   RUNG wire#w3
      R_Coil( "3号梯七段数码管f" )
   END_RUNG
   RUNG wire#w3
      S_Coil( "3号梯七段数码管g" )
   END_RUNG
   RUNG wire#w3
      R_Coil( "3号梯七段数码管h" )
   END_RUNG
   RUNG wire#w3
      R_Coil( "3号梯七段数码管i" )
   END_RUNG
   RUNG wire#w3
      R_Coil( "3号梯七段数码管j" )
   END_RUNG
   RUNG wire#w3
      R_Coil( "3号梯七段数码管k" )
   END_RUNG
   RUNG wire#w3
      R_Coil( "3号梯七段数码管l" )
   END_RUNG
   RUNG wire#w3
      R_Coil( "3号梯七段数码管m" )
   END_RUNG
   RUNG wire#w3
      R_Coil( "3号梯七段数码管n" )
   END_RUNG
   RUNG wire#powerrail
      { S7_Templates := "SrcType := Int" } EQ_Contact(in1 := "3号梯当前楼层数", in2 := 4)
      wire#w4
      R_Coil( "3号梯七段数码管a" )
   END_RUNG
   RUNG wire#w4
      S_Coil( "3号梯七段数码管b" )
   END_RUNG
   RUNG wire#w4
      S_Coil( "3号梯七段数码管c" )
   END_RUNG
   RUNG wire#w4
      R_Coil( "3号梯七段数码管d" )
   END_RUNG
   RUNG wire#w4
      R_Coil( "3号梯七段数码管e" )
   END_RUNG
   RUNG wire#w4
      S_Coil( "3号梯七段数码管f" )
   END_RUNG
   RUNG wire#w4
      S_Coil( "3号梯七段数码管g" )
   END_RUNG
   RUNG wire#w4
      R_Coil( "3号梯七段数码管h" )
   END_RUNG
   RUNG wire#w4
      R_Coil( "3号梯七段数码管i" )
   END_RUNG
   RUNG wire#w4
      R_Coil( "3号梯七段数码管j" )
   END_RUNG
   RUNG wire#w4
      R_Coil( "3号梯七段数码管k" )
   END_RUNG
   RUNG wire#w4
      R_Coil( "3号梯七段数码管l" )
   END_RUNG
   RUNG wire#w4
      R_Coil( "3号梯七段数码管m" )
   END_RUNG
   RUNG wire#w4
      R_Coil( "3号梯七段数码管n" )
   END_RUNG
   RUNG wire#powerrail
      { S7_Templates := "SrcType := Int" } EQ_Contact(in1 := "3号梯当前楼层数", in2 := 5)
      wire#w5
      S_Coil( "3号梯七段数码管a" )
   END_RUNG
   RUNG wire#w5
      R_Coil( "3号梯七段数码管b" )
   END_RUNG
   RUNG wire#w5
      S_Coil( "3号梯七段数码管c" )
   END_RUNG
   RUNG wire#w5
      S_Coil( "3号梯七段数码管d" )
   END_RUNG
   RUNG wire#w5
      R_Coil( "3号梯七段数码管e" )
   END_RUNG
   RUNG wire#w5
      S_Coil( "3号梯七段数码管f" )
   END_RUNG
   RUNG wire#w5
      S_Coil( "3号梯七段数码管g" )
   END_RUNG
   RUNG wire#w5
      R_Coil( "3号梯七段数码管h" )
   END_RUNG
   RUNG wire#w5
      R_Coil( "3号梯七段数码管i" )
   END_RUNG
   RUNG wire#w5
      R_Coil( "3号梯七段数码管j" )
   END_RUNG
   RUNG wire#w5
      R_Coil( "3号梯七段数码管k" )
   END_RUNG
   RUNG wire#w5
      R_Coil( "3号梯七段数码管l" )
   END_RUNG
   RUNG wire#w5
      R_Coil( "3号梯七段数码管m" )
   END_RUNG
   RUNG wire#w5
      R_Coil( "3号梯七段数码管n" )
   END_RUNG
   RUNG wire#powerrail
      { S7_Templates := "SrcType := Int" } EQ_Contact(in1 := "3号梯当前楼层数", in2 := 6)
      wire#w6
      S_Coil( "3号梯七段数码管a" )
   END_RUNG
   RUNG wire#w6
      R_Coil( "3号梯七段数码管b" )
   END_RUNG
   RUNG wire#w6
      S_Coil( "3号梯七段数码管c" )
   END_RUNG
   RUNG wire#w6
      S_Coil( "3号梯七段数码管d" )
   END_RUNG
   RUNG wire#w6
      S_Coil( "3号梯七段数码管e" )
   END_RUNG
   RUNG wire#w6
      S_Coil( "3号梯七段数码管f" )
   END_RUNG
   RUNG wire#w6
      S_Coil( "3号梯七段数码管g" )
   END_RUNG
   RUNG wire#w6
      R_Coil( "3号梯七段数码管h" )
   END_RUNG
   RUNG wire#w6
      R_Coil( "3号梯七段数码管i" )
   END_RUNG
   RUNG wire#w6
      R_Coil( "3号梯七段数码管j" )
   END_RUNG
   RUNG wire#w6
      R_Coil( "3号梯七段数码管k" )
   END_RUNG
   RUNG wire#w6
      R_Coil( "3号梯七段数码管l" )
   END_RUNG
   RUNG wire#w6
      R_Coil( "3号梯七段数码管m" )
   END_RUNG
   RUNG wire#w6
      R_Coil( "3号梯七段数码管n" )
   END_RUNG
   RUNG wire#powerrail
      { S7_Templates := "SrcType := Int" } EQ_Contact(in1 := "3号梯当前楼层数", in2 := 7)
      wire#w7
      S_Coil( "3号梯七段数码管a" )
   END_RUNG
   RUNG wire#w7
      S_Coil( "3号梯七段数码管b" )
   END_RUNG
   RUNG wire#w7
      S_Coil( "3号梯七段数码管c" )
   END_RUNG
   RUNG wire#w7
      R_Coil( "3号梯七段数码管d" )
   END_RUNG
   RUNG wire#w7
      R_Coil( "3号梯七段数码管e" )
   END_RUNG
   RUNG wire#w7
      R_Coil( "3号梯七段数码管f" )
   END_RUNG
   RUNG wire#w7
      R_Coil( "3号梯七段数码管g" )
   END_RUNG
   RUNG wire#w7
      R_Coil( "3号梯七段数码管h" )
   END_RUNG
   RUNG wire#w7
      R_Coil( "3号梯七段数码管i" )
   END_RUNG
   RUNG wire#w7
      R_Coil( "3号梯七段数码管j" )
   END_RUNG
   RUNG wire#w7
      R_Coil( "3号梯七段数码管k" )
   END_RUNG
   RUNG wire#w7
      R_Coil( "3号梯七段数码管l" )
   END_RUNG
   RUNG wire#w7
      R_Coil( "3号梯七段数码管m" )
   END_RUNG
   RUNG wire#w7
      R_Coil( "3号梯七段数码管n" )
   END_RUNG
   RUNG wire#powerrail
      { S7_Templates := "SrcType := Int" } EQ_Contact(in1 := "3号梯当前楼层数", in2 := 8)
      wire#w8
      S_Coil( "3号梯七段数码管a" )
   END_RUNG
   RUNG wire#w8
      S_Coil( "3号梯七段数码管b" )
   END_RUNG
   RUNG wire#w8
      S_Coil( "3号梯七段数码管c" )
   END_RUNG
   RUNG wire#w8
      S_Coil( "3号梯七段数码管d" )
   END_RUNG
   RUNG wire#w8
      S_Coil( "3号梯七段数码管e" )
   END_RUNG
   RUNG wire#w8
      S_Coil( "3号梯七段数码管f" )
   END_RUNG
   RUNG wire#w8
      S_Coil( "3号梯七段数码管g" )
   END_RUNG
   RUNG wire#w8
      R_Coil( "3号梯七段数码管h" )
   END_RUNG
   RUNG wire#w8
      R_Coil( "3号梯七段数码管i" )
   END_RUNG
   RUNG wire#w8
      R_Coil( "3号梯七段数码管j" )
   END_RUNG
   RUNG wire#w8
      R_Coil( "3号梯七段数码管k" )
   END_RUNG
   RUNG wire#w8
      R_Coil( "3号梯七段数码管l" )
   END_RUNG
   RUNG wire#w8
      R_Coil( "3号梯七段数码管m" )
   END_RUNG
   RUNG wire#w8
      R_Coil( "3号梯七段数码管n" )
   END_RUNG
   RUNG wire#powerrail
      { S7_Templates := "SrcType := Int" } EQ_Contact(in1 := "3号梯当前楼层数", in2 := 9)
      wire#w9
      S_Coil( "3号梯七段数码管a" )
   END_RUNG
   RUNG wire#w9
      S_Coil( "3号梯七段数码管b" )
   END_RUNG
   RUNG wire#w9
      S_Coil( "3号梯七段数码管c" )
   END_RUNG
   RUNG wire#w9
      S_Coil( "3号梯七段数码管d" )
   END_RUNG
   RUNG wire#w9
      R_Coil( "3号梯七段数码管e" )
   END_RUNG
   RUNG wire#w9
      S_Coil( "3号梯七段数码管f" )
   END_RUNG
   RUNG wire#w9
      S_Coil( "3号梯七段数码管g" )
   END_RUNG
   RUNG wire#w9
      R_Coil( "3号梯七段数码管h" )
   END_RUNG
   RUNG wire#w9
      R_Coil( "3号梯七段数码管i" )
   END_RUNG
   RUNG wire#w9
      R_Coil( "3号梯七段数码管j" )
   END_RUNG
   RUNG wire#w9
      R_Coil( "3号梯七段数码管k" )
   END_RUNG
   RUNG wire#w9
      R_Coil( "3号梯七段数码管l" )
   END_RUNG
   RUNG wire#w9
      R_Coil( "3号梯七段数码管m" )
   END_RUNG
   RUNG wire#w9
      R_Coil( "3号梯七段数码管n" )
   END_RUNG
   RUNG wire#powerrail
      { S7_Templates := "SrcType := Int" } EQ_Contact(in1 := "3号梯当前楼层数", in2 := 10)
      wire#w10
      S_Coil( "3号梯七段数码管a" )
   END_RUNG
   RUNG wire#w10
      S_Coil( "3号梯七段数码管b" )
   END_RUNG
   RUNG wire#w10
      S_Coil( "3号梯七段数码管c" )
   END_RUNG
   RUNG wire#w10
      S_Coil( "3号梯七段数码管d" )
   END_RUNG
   RUNG wire#w10
      S_Coil( "3号梯七段数码管e" )
   END_RUNG
   RUNG wire#w10
      S_Coil( "3号梯七段数码管f" )
   END_RUNG
   RUNG wire#w10
      R_Coil( "3号梯七段数码管g" )
   END_RUNG
   RUNG wire#w10
      R_Coil( "3号梯七段数码管h" )
   END_RUNG
   RUNG wire#w10
      S_Coil( "3号梯七段数码管i" )
   END_RUNG
   RUNG wire#w10
      S_Coil( "3号梯七段数码管j" )
   END_RUNG
   RUNG wire#w10
      R_Coil( "3号梯七段数码管k" )
   END_RUNG
   RUNG wire#w10
      R_Coil( "3号梯七段数码管l" )
   END_RUNG
   RUNG wire#w10
      R_Coil( "3号梯七段数码管m" )
   END_RUNG
   RUNG wire#w10
      R_Coil( "3号梯七段数码管n" )
   END_RUNG
   // the same network as SCL:
   IF "3号梯当前楼层数" = 1 THEN
       "3号梯七段数码管a" := FALSE;
       "3号梯七段数码管b" := TRUE;
       "3号梯七段数码管c" := TRUE;
       "3号梯七段数码管d" := FALSE;
       "3号梯七段数码管e" := FALSE;
       "3号梯七段数码管f" := FALSE;
       "3号梯七段数码管g" := FALSE;
       "3号梯七段数码管h" := FALSE;
       "3号梯七段数码管i" := FALSE;
       "3号梯七段数码管j" := FALSE;
       "3号梯七段数码管k" := FALSE;
       "3号梯七段数码管l" := FALSE;
       "3号梯七段数码管m" := FALSE;
       "3号梯七段数码管n" := FALSE;
   END_IF;
   IF "3号梯当前楼层数" = 2 THEN
       "3号梯七段数码管a" := TRUE;
       "3号梯七段数码管b" := TRUE;
       "3号梯七段数码管c" := FALSE;
       "3号梯七段数码管d" := TRUE;
       "3号梯七段数码管e" := TRUE;
       "3号梯七段数码管f" := FALSE;
       "3号梯七段数码管g" := TRUE;
       "3号梯七段数码管h" := FALSE;
       "3号梯七段数码管i" := FALSE;
       "3号梯七段数码管j" := FALSE;
       "3号梯七段数码管k" := FALSE;
       "3号梯七段数码管l" := FALSE;
       "3号梯七段数码管m" := FALSE;
       "3号梯七段数码管n" := FALSE;
   END_IF;
   IF "3号梯当前楼层数" = 3 THEN
       "3号梯七段数码管a" := TRUE;
       "3号梯七段数码管b" := TRUE;
       "3号梯七段数码管c" := TRUE;
       "3号梯七段数码管d" := TRUE;
       "3号梯七段数码管e" := FALSE;
       "3号梯七段数码管f" := FALSE;
       "3号梯七段数码管g" := TRUE;
       "3号梯七段数码管h" := FALSE;
       "3号梯七段数码管i" := FALSE;
       "3号梯七段数码管j" := FALSE;
       "3号梯七段数码管k" := FALSE;
       "3号梯七段数码管l" := FALSE;
       "3号梯七段数码管m" := FALSE;
       "3号梯七段数码管n" := FALSE;
   END_IF;
   IF "3号梯当前楼层数" = 4 THEN
       "3号梯七段数码管a" := FALSE;
       "3号梯七段数码管b" := TRUE;
       "3号梯七段数码管c" := TRUE;
       "3号梯七段数码管d" := FALSE;
       "3号梯七段数码管e" := FALSE;
       "3号梯七段数码管f" := TRUE;
       "3号梯七段数码管g" := TRUE;
       "3号梯七段数码管h" := FALSE;
       "3号梯七段数码管i" := FALSE;
       "3号梯七段数码管j" := FALSE;
       "3号梯七段数码管k" := FALSE;
       "3号梯七段数码管l" := FALSE;
       "3号梯七段数码管m" := FALSE;
       "3号梯七段数码管n" := FALSE;
   END_IF;
   IF "3号梯当前楼层数" = 5 THEN
       "3号梯七段数码管a" := TRUE;
       "3号梯七段数码管b" := FALSE;
       "3号梯七段数码管c" := TRUE;
       "3号梯七段数码管d" := TRUE;
       "3号梯七段数码管e" := FALSE;
       "3号梯七段数码管f" := TRUE;
       "3号梯七段数码管g" := TRUE;
       "3号梯七段数码管h" := FALSE;
       "3号梯七段数码管i" := FALSE;
       "3号梯七段数码管j" := FALSE;
       "3号梯七段数码管k" := FALSE;
       "3号梯七段数码管l" := FALSE;
       "3号梯七段数码管m" := FALSE;
       "3号梯七段数码管n" := FALSE;
   END_IF;
   IF "3号梯当前楼层数" = 6 THEN
       "3号梯七段数码管a" := TRUE;
       "3号梯七段数码管b" := FALSE;
       "3号梯七段数码管c" := TRUE;
       "3号梯七段数码管d" := TRUE;
       "3号梯七段数码管e" := TRUE;
       "3号梯七段数码管f" := TRUE;
       "3号梯七段数码管g" := TRUE;
       "3号梯七段数码管h" := FALSE;
       "3号梯七段数码管i" := FALSE;
       "3号梯七段数码管j" := FALSE;
       "3号梯七段数码管k" := FALSE;
       "3号梯七段数码管l" := FALSE;
       "3号梯七段数码管m" := FALSE;
       "3号梯七段数码管n" := FALSE;
   END_IF;
   IF "3号梯当前楼层数" = 7 THEN
       "3号梯七段数码管a" := TRUE;
       "3号梯七段数码管b" := TRUE;
       "3号梯七段数码管c" := TRUE;
       "3号梯七段数码管d" := FALSE;
       "3号梯七段数码管e" := FALSE;
       "3号梯七段数码管f" := FALSE;
       "3号梯七段数码管g" := FALSE;
       "3号梯七段数码管h" := FALSE;
       "3号梯七段数码管i" := FALSE;
       "3号梯七段数码管j" := FALSE;
       "3号梯七段数码管k" := FALSE;
       "3号梯七段数码管l" := FALSE;
       "3号梯七段数码管m" := FALSE;
       "3号梯七段数码管n" := FALSE;
   END_IF;
   IF "3号梯当前楼层数" = 8 THEN
       "3号梯七段数码管a" := TRUE;
       "3号梯七段数码管b" := TRUE;
       "3号梯七段数码管c" := TRUE;
       "3号梯七段数码管d" := TRUE;
       "3号梯七段数码管e" := TRUE;
       "3号梯七段数码管f" := TRUE;
       "3号梯七段数码管g" := TRUE;
       "3号梯七段数码管h" := FALSE;
       "3号梯七段数码管i" := FALSE;
       "3号梯七段数码管j" := FALSE;
       "3号梯七段数码管k" := FALSE;
       "3号梯七段数码管l" := FALSE;
       "3号梯七段数码管m" := FALSE;
       "3号梯七段数码管n" := FALSE;
   END_IF;
   IF "3号梯当前楼层数" = 9 THEN
       "3号梯七段数码管a" := TRUE;
       "3号梯七段数码管b" := TRUE;
       "3号梯七段数码管c" := TRUE;
       "3号梯七段数码管d" := TRUE;
       "3号梯七段数码管e" := FALSE;
       "3号梯七段数码管f" := TRUE;
       "3号梯七段数码管g" := TRUE;
       "3号梯七段数码管h" := FALSE;
       "3号梯七段数码管i" := FALSE;
       "3号梯七段数码管j" := FALSE;
       "3号梯七段数码管k" := FALSE;
       "3号梯七段数码管l" := FALSE;
       "3号梯七段数码管m" := FALSE;
       "3号梯七段数码管n" := FALSE;
   END_IF;
   IF "3号梯当前楼层数" = 10 THEN
       "3号梯七段数码管a" := TRUE;
       "3号梯七段数码管b" := TRUE;
       "3号梯七段数码管c" := TRUE;
       "3号梯七段数码管d" := TRUE;
       "3号梯七段数码管e" := TRUE;
       "3号梯七段数码管f" := TRUE;
       "3号梯七段数码管g" := FALSE;
       "3号梯七段数码管h" := FALSE;
       "3号梯七段数码管i" := TRUE;
       "3号梯七段数码管j" := TRUE;
       "3号梯七段数码管k" := FALSE;
       "3号梯七段数码管l" := FALSE;
       "3号梯七段数码管m" := FALSE;
       "3号梯七段数码管n" := FALSE;
   END_IF;
END_REGION

REGION Network 2: 上下行指示灯
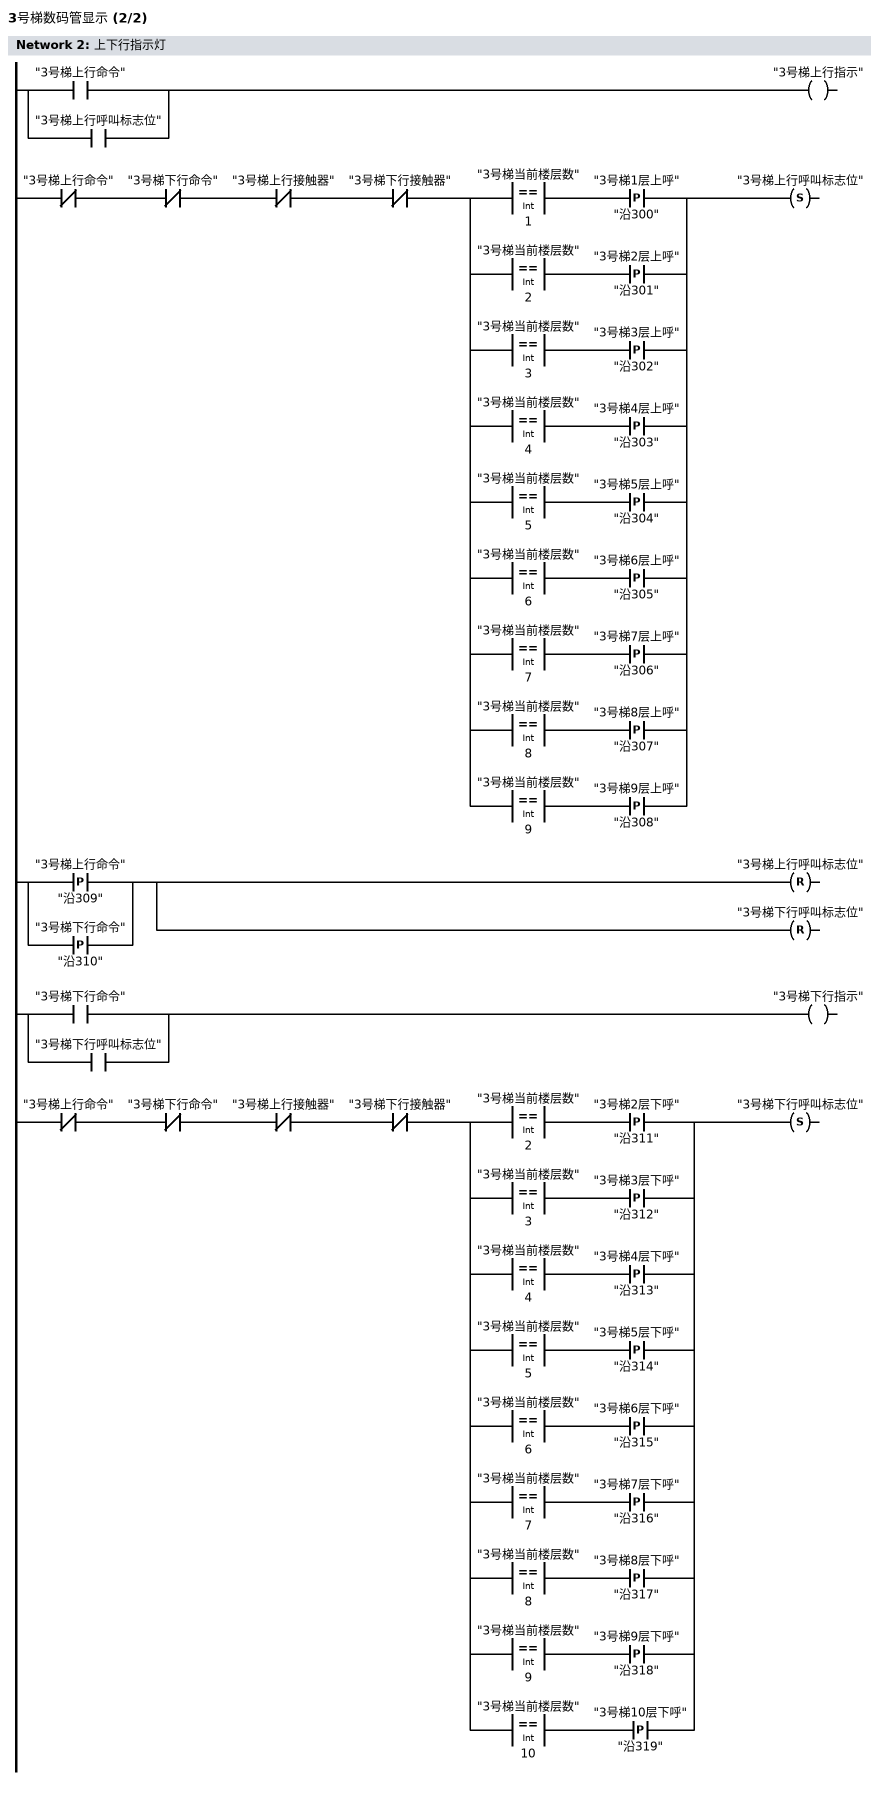
   RUNG wire#powerrail
      Contact( "3号梯上行命令" )
      wire#w1
      Coil( "3号梯上行指示" )
   END_RUNG
   RUNG wire#powerrail
      Contact( "3号梯上行呼叫标志位" )
   END_RUNG wire#w1
   RUNG wire#powerrail
      I_Contact( "3号梯上行命令" )
      I_Contact( "3号梯下行命令" )
      I_Contact( "3号梯上行接触器" )
      I_Contact( "3号梯下行接触器" )
      wire#w2
      { S7_Templates := "SrcType := Int" } EQ_Contact(in1 := "3号梯当前楼层数", in2 := 1)
      P_Contact(operand := "3号梯1层上呼", bit := "沿300")
      wire#w3
      S_Coil( "3号梯上行呼叫标志位" )
   END_RUNG
   RUNG wire#w2
      { S7_Templates := "SrcType := Int" } EQ_Contact(in1 := "3号梯当前楼层数", in2 := 2)
      P_Contact(operand := "3号梯2层上呼", bit := "沿301")
   END_RUNG wire#w3
   RUNG wire#w2
      { S7_Templates := "SrcType := Int" } EQ_Contact(in1 := "3号梯当前楼层数", in2 := 3)
      P_Contact(operand := "3号梯3层上呼", bit := "沿302")
   END_RUNG wire#w3
   RUNG wire#w2
      { S7_Templates := "SrcType := Int" } EQ_Contact(in1 := "3号梯当前楼层数", in2 := 4)
      P_Contact(operand := "3号梯4层上呼", bit := "沿303")
   END_RUNG wire#w3
   RUNG wire#w2
      { S7_Templates := "SrcType := Int" } EQ_Contact(in1 := "3号梯当前楼层数", in2 := 5)
      P_Contact(operand := "3号梯5层上呼", bit := "沿304")
   END_RUNG wire#w3
   RUNG wire#w2
      { S7_Templates := "SrcType := Int" } EQ_Contact(in1 := "3号梯当前楼层数", in2 := 6)
      P_Contact(operand := "3号梯6层上呼", bit := "沿305")
   END_RUNG wire#w3
   RUNG wire#w2
      { S7_Templates := "SrcType := Int" } EQ_Contact(in1 := "3号梯当前楼层数", in2 := 7)
      P_Contact(operand := "3号梯7层上呼", bit := "沿306")
   END_RUNG wire#w3
   RUNG wire#w2
      { S7_Templates := "SrcType := Int" } EQ_Contact(in1 := "3号梯当前楼层数", in2 := 8)
      P_Contact(operand := "3号梯8层上呼", bit := "沿307")
   END_RUNG wire#w3
   RUNG wire#w2
      { S7_Templates := "SrcType := Int" } EQ_Contact(in1 := "3号梯当前楼层数", in2 := 9)
      P_Contact(operand := "3号梯9层上呼", bit := "沿308")
   END_RUNG wire#w3
   RUNG wire#powerrail
      P_Contact(operand := "3号梯上行命令", bit := "沿309")
      wire#w4
      R_Coil( "3号梯上行呼叫标志位" )
   END_RUNG
   RUNG wire#powerrail
      P_Contact(operand := "3号梯下行命令", bit := "沿310")
   END_RUNG wire#w4
   RUNG wire#w4
      R_Coil( "3号梯下行呼叫标志位" )
   END_RUNG
   RUNG wire#powerrail
      Contact( "3号梯下行命令" )
      wire#w5
      Coil( "3号梯下行指示" )
   END_RUNG
   RUNG wire#powerrail
      Contact( "3号梯下行呼叫标志位" )
   END_RUNG wire#w5
   RUNG wire#powerrail
      I_Contact( "3号梯上行命令" )
      I_Contact( "3号梯下行命令" )
      I_Contact( "3号梯上行接触器" )
      I_Contact( "3号梯下行接触器" )
      wire#w6
      { S7_Templates := "SrcType := Int" } EQ_Contact(in1 := "3号梯当前楼层数", in2 := 2)
      P_Contact(operand := "3号梯2层下呼", bit := "沿311")
      wire#w7
      S_Coil( "3号梯下行呼叫标志位" )
   END_RUNG
   RUNG wire#w6
      { S7_Templates := "SrcType := Int" } EQ_Contact(in1 := "3号梯当前楼层数", in2 := 3)
      P_Contact(operand := "3号梯3层下呼", bit := "沿312")
   END_RUNG wire#w7
   RUNG wire#w6
      { S7_Templates := "SrcType := Int" } EQ_Contact(in1 := "3号梯当前楼层数", in2 := 4)
      P_Contact(operand := "3号梯4层下呼", bit := "沿313")
   END_RUNG wire#w7
   RUNG wire#w6
      { S7_Templates := "SrcType := Int" } EQ_Contact(in1 := "3号梯当前楼层数", in2 := 5)
      P_Contact(operand := "3号梯5层下呼", bit := "沿314")
   END_RUNG wire#w7
   RUNG wire#w6
      { S7_Templates := "SrcType := Int" } EQ_Contact(in1 := "3号梯当前楼层数", in2 := 6)
      P_Contact(operand := "3号梯6层下呼", bit := "沿315")
   END_RUNG wire#w7
   RUNG wire#w6
      { S7_Templates := "SrcType := Int" } EQ_Contact(in1 := "3号梯当前楼层数", in2 := 7)
      P_Contact(operand := "3号梯7层下呼", bit := "沿316")
   END_RUNG wire#w7
   RUNG wire#w6
      { S7_Templates := "SrcType := Int" } EQ_Contact(in1 := "3号梯当前楼层数", in2 := 8)
      P_Contact(operand := "3号梯8层下呼", bit := "沿317")
   END_RUNG wire#w7
   RUNG wire#w6
      { S7_Templates := "SrcType := Int" } EQ_Contact(in1 := "3号梯当前楼层数", in2 := 9)
      P_Contact(operand := "3号梯9层下呼", bit := "沿318")
   END_RUNG wire#w7
   RUNG wire#w6
      { S7_Templates := "SrcType := Int" } EQ_Contact(in1 := "3号梯当前楼层数", in2 := 10)
      P_Contact(operand := "3号梯10层下呼", bit := "沿319")
   END_RUNG wire#w7
   // the same network as SCL:
   "3号梯上行指示" := "3号梯上行命令" OR "3号梯上行呼叫标志位";
   #_w1 := NOT "3号梯上行命令" AND NOT "3号梯下行命令" AND NOT "3号梯上行接触器" AND NOT "3号梯下行接触器" AND ("3号梯当前楼层数" = 1) AND "3号梯1层上呼" AND NOT "沿300";   // rising edge of "3号梯1层上呼"
   "沿300" := "3号梯1层上呼";
   #_w2 := NOT "3号梯上行命令" AND NOT "3号梯下行命令" AND NOT "3号梯上行接触器" AND NOT "3号梯下行接触器" AND ("3号梯当前楼层数" = 2) AND "3号梯2层上呼" AND NOT "沿301";   // rising edge of "3号梯2层上呼"
   "沿301" := "3号梯2层上呼";
   #_w3 := NOT "3号梯上行命令" AND NOT "3号梯下行命令" AND NOT "3号梯上行接触器" AND NOT "3号梯下行接触器" AND ("3号梯当前楼层数" = 3) AND "3号梯3层上呼" AND NOT "沿302";   // rising edge of "3号梯3层上呼"
   "沿302" := "3号梯3层上呼";
   #_w4 := NOT "3号梯上行命令" AND NOT "3号梯下行命令" AND NOT "3号梯上行接触器" AND NOT "3号梯下行接触器" AND ("3号梯当前楼层数" = 4) AND "3号梯4层上呼" AND NOT "沿303";   // rising edge of "3号梯4层上呼"
   "沿303" := "3号梯4层上呼";
   #_w5 := NOT "3号梯上行命令" AND NOT "3号梯下行命令" AND NOT "3号梯上行接触器" AND NOT "3号梯下行接触器" AND ("3号梯当前楼层数" = 5) AND "3号梯5层上呼" AND NOT "沿304";   // rising edge of "3号梯5层上呼"
   "沿304" := "3号梯5层上呼";
   #_w6 := NOT "3号梯上行命令" AND NOT "3号梯下行命令" AND NOT "3号梯上行接触器" AND NOT "3号梯下行接触器" AND ("3号梯当前楼层数" = 6) AND "3号梯6层上呼" AND NOT "沿305";   // rising edge of "3号梯6层上呼"
   "沿305" := "3号梯6层上呼";
   #_w7 := NOT "3号梯上行命令" AND NOT "3号梯下行命令" AND NOT "3号梯上行接触器" AND NOT "3号梯下行接触器" AND ("3号梯当前楼层数" = 7) AND "3号梯7层上呼" AND NOT "沿306";   // rising edge of "3号梯7层上呼"
   "沿306" := "3号梯7层上呼";
   #_w8 := NOT "3号梯上行命令" AND NOT "3号梯下行命令" AND NOT "3号梯上行接触器" AND NOT "3号梯下行接触器" AND ("3号梯当前楼层数" = 8) AND "3号梯8层上呼" AND NOT "沿307";   // rising edge of "3号梯8层上呼"
   "沿307" := "3号梯8层上呼";
   #_w9 := NOT "3号梯上行命令" AND NOT "3号梯下行命令" AND NOT "3号梯上行接触器" AND NOT "3号梯下行接触器" AND ("3号梯当前楼层数" = 9) AND "3号梯9层上呼" AND NOT "沿308";   // rising edge of "3号梯9层上呼"
   "沿308" := "3号梯9层上呼";
   IF #_w1 OR #_w2 OR #_w3 OR #_w4 OR #_w5 OR #_w6 OR #_w7 OR #_w8 OR #_w9 THEN "3号梯上行呼叫标志位" := TRUE; END_IF;
   #_w10 := "3号梯上行命令" AND NOT "沿309";   // rising edge of "3号梯上行命令"
   "沿309" := "3号梯上行命令";
   #_w11 := "3号梯下行命令" AND NOT "沿310";   // rising edge of "3号梯下行命令"
   "沿310" := "3号梯下行命令";
   IF #_w10 OR #_w11 THEN
       "3号梯上行呼叫标志位" := FALSE;
       "3号梯下行呼叫标志位" := FALSE;
   END_IF;
   "3号梯下行指示" := "3号梯下行命令" OR "3号梯下行呼叫标志位";
   #_w12 := NOT "3号梯上行命令" AND NOT "3号梯下行命令" AND NOT "3号梯上行接触器" AND NOT "3号梯下行接触器" AND ("3号梯当前楼层数" = 2) AND "3号梯2层下呼" AND NOT "沿311";   // rising edge of "3号梯2层下呼"
   "沿311" := "3号梯2层下呼";
   #_w13 := NOT "3号梯上行命令" AND NOT "3号梯下行命令" AND NOT "3号梯上行接触器" AND NOT "3号梯下行接触器" AND ("3号梯当前楼层数" = 3) AND "3号梯3层下呼" AND NOT "沿312";   // rising edge of "3号梯3层下呼"
   "沿312" := "3号梯3层下呼";
   #_w14 := NOT "3号梯上行命令" AND NOT "3号梯下行命令" AND NOT "3号梯上行接触器" AND NOT "3号梯下行接触器" AND ("3号梯当前楼层数" = 4) AND "3号梯4层下呼" AND NOT "沿313";   // rising edge of "3号梯4层下呼"
   "沿313" := "3号梯4层下呼";
   #_w15 := NOT "3号梯上行命令" AND NOT "3号梯下行命令" AND NOT "3号梯上行接触器" AND NOT "3号梯下行接触器" AND ("3号梯当前楼层数" = 5) AND "3号梯5层下呼" AND NOT "沿314";   // rising edge of "3号梯5层下呼"
   "沿314" := "3号梯5层下呼";
   #_w16 := NOT "3号梯上行命令" AND NOT "3号梯下行命令" AND NOT "3号梯上行接触器" AND NOT "3号梯下行接触器" AND ("3号梯当前楼层数" = 6) AND "3号梯6层下呼" AND NOT "沿315";   // rising edge of "3号梯6层下呼"
   "沿315" := "3号梯6层下呼";
   #_w17 := NOT "3号梯上行命令" AND NOT "3号梯下行命令" AND NOT "3号梯上行接触器" AND NOT "3号梯下行接触器" AND ("3号梯当前楼层数" = 7) AND "3号梯7层下呼" AND NOT "沿316";   // rising edge of "3号梯7层下呼"
   "沿316" := "3号梯7层下呼";
   #_w18 := NOT "3号梯上行命令" AND NOT "3号梯下行命令" AND NOT "3号梯上行接触器" AND NOT "3号梯下行接触器" AND ("3号梯当前楼层数" = 8) AND "3号梯8层下呼" AND NOT "沿317";   // rising edge of "3号梯8层下呼"
   "沿317" := "3号梯8层下呼";
   #_w19 := NOT "3号梯上行命令" AND NOT "3号梯下行命令" AND NOT "3号梯上行接触器" AND NOT "3号梯下行接触器" AND ("3号梯当前楼层数" = 9) AND "3号梯9层下呼" AND NOT "沿318";   // rising edge of "3号梯9层下呼"
   "沿318" := "3号梯9层下呼";
   #_w20 := NOT "3号梯上行命令" AND NOT "3号梯下行命令" AND NOT "3号梯上行接触器" AND NOT "3号梯下行接触器" AND ("3号梯当前楼层数" = 10) AND "3号梯10层下呼" AND NOT "沿319";   // rising edge of "3号梯10层下呼"
   "沿319" := "3号梯10层下呼";
   IF #_w12 OR #_w13 OR #_w14 OR #_w15 OR #_w16 OR #_w17 OR #_w18 OR #_w19 OR #_w20 THEN
       "3号梯下行呼叫标志位" := TRUE;
   END_IF;
END_REGION
END_FUNCTION

FUNCTION "3号电梯初始化" : Void   // FC24, LAD
{ S7_Optimized_Access := 'TRUE' }
VERSION : 0.1
   VAR_TEMP   // added for the SCL form of the ladder/FBD networks
      _w1 : Bool;
   END_VAR
BEGIN

REGION Network 1: 上下行初始化选择
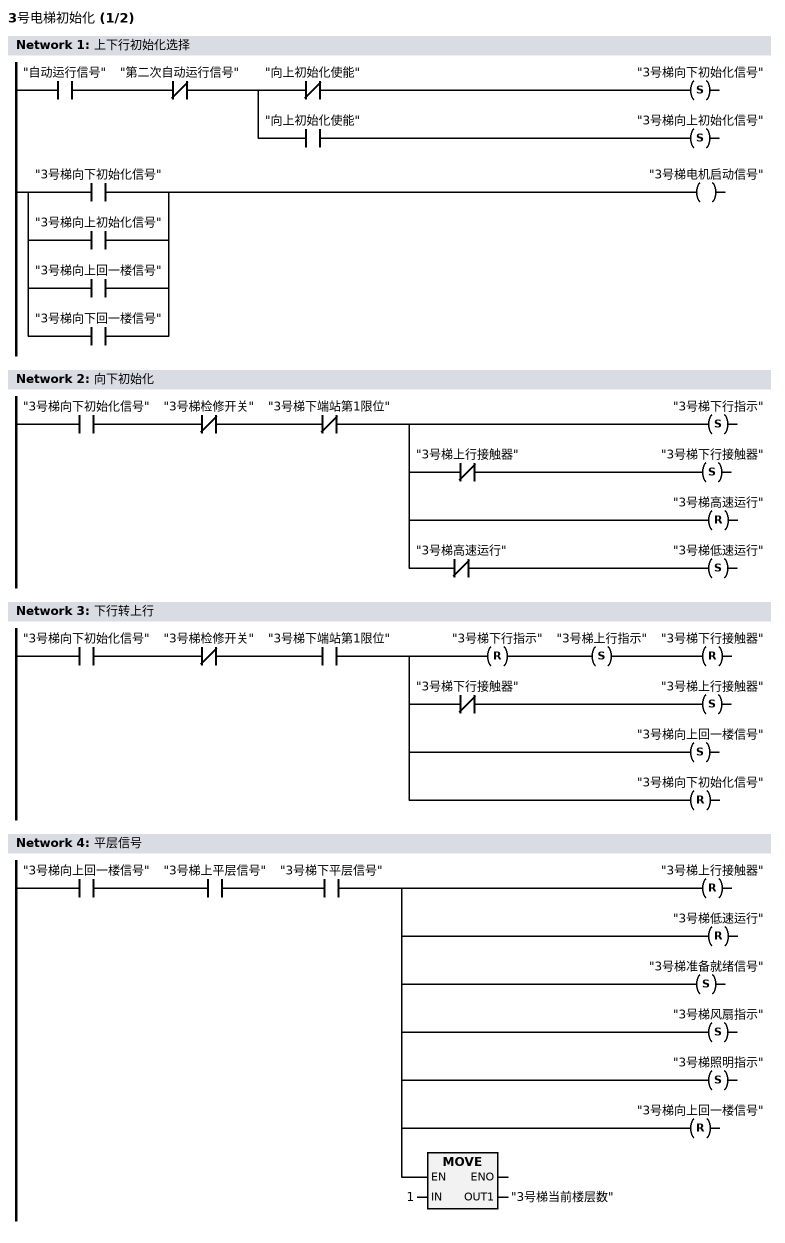
   RUNG wire#powerrail
      Contact( "自动运行信号" )
      I_Contact( "第二次自动运行信号" )
      wire#w1
      I_Contact( "向上初始化使能" )
      S_Coil( "3号梯向下初始化信号" )
   END_RUNG
   RUNG wire#w1
      Contact( "向上初始化使能" )
      S_Coil( "3号梯向上初始化信号" )
   END_RUNG
   RUNG wire#powerrail
      Contact( "3号梯向下初始化信号" )
      wire#w2
      Coil( "3号梯电机启动信号" )
   END_RUNG
   RUNG wire#powerrail
      Contact( "3号梯向上初始化信号" )
   END_RUNG wire#w2
   RUNG wire#powerrail
      Contact( "3号梯向上回一楼信号" )
   END_RUNG wire#w2
   RUNG wire#powerrail
      Contact( "3号梯向下回一楼信号" )
   END_RUNG wire#w2
   // the same network as SCL:
   #_w1 := "自动运行信号" AND NOT "第二次自动运行信号";
   IF #_w1 AND NOT "向上初始化使能" THEN "3号梯向下初始化信号" := TRUE; END_IF;
   IF #_w1 AND "向上初始化使能" THEN "3号梯向上初始化信号" := TRUE; END_IF;
   "3号梯电机启动信号" := "3号梯向下初始化信号" OR "3号梯向上初始化信号" OR "3号梯向上回一楼信号" OR "3号梯向下回一楼信号";
END_REGION

REGION Network 2: 向下初始化
   RUNG wire#powerrail
      Contact( "3号梯向下初始化信号" )
      I_Contact( "3号梯检修开关" )
      I_Contact( "3号梯下端站第1限位" )
      wire#w1
      S_Coil( "3号梯下行指示" )
   END_RUNG
   RUNG wire#w1
      I_Contact( "3号梯上行接触器" )
      S_Coil( "3号梯下行接触器" )
   END_RUNG
   RUNG wire#w1
      R_Coil( "3号梯高速运行" )
   END_RUNG
   RUNG wire#w1
      I_Contact( "3号梯高速运行" )
      S_Coil( "3号梯低速运行" )
   END_RUNG
   // the same network as SCL:
   #_w1 := "3号梯向下初始化信号" AND NOT "3号梯检修开关" AND NOT "3号梯下端站第1限位";
   IF #_w1 THEN "3号梯下行指示" := TRUE; END_IF;
   IF #_w1 AND NOT "3号梯上行接触器" THEN "3号梯下行接触器" := TRUE; END_IF;
   IF #_w1 THEN "3号梯高速运行" := FALSE; END_IF;
   IF #_w1 AND NOT "3号梯高速运行" THEN "3号梯低速运行" := TRUE; END_IF;
END_REGION

REGION Network 3: 下行转上行
   RUNG wire#powerrail
      Contact( "3号梯向下初始化信号" )
      I_Contact( "3号梯检修开关" )
      Contact( "3号梯下端站第1限位" )
      wire#w1
      R_Coil( "3号梯下行指示" )
      S_Coil( "3号梯上行指示" )
      R_Coil( "3号梯下行接触器" )
   END_RUNG
   RUNG wire#w1
      I_Contact( "3号梯下行接触器" )
      S_Coil( "3号梯上行接触器" )
   END_RUNG
   RUNG wire#w1
      S_Coil( "3号梯向上回一楼信号" )
   END_RUNG
   RUNG wire#w1
      R_Coil( "3号梯向下初始化信号" )
   END_RUNG
   // the same network as SCL:
   #_w1 := "3号梯向下初始化信号" AND NOT "3号梯检修开关" AND "3号梯下端站第1限位";
   IF #_w1 THEN
       "3号梯下行指示" := FALSE;
       "3号梯上行指示" := TRUE;
       "3号梯下行接触器" := FALSE;
   END_IF;
   IF #_w1 AND NOT "3号梯下行接触器" THEN "3号梯上行接触器" := TRUE; END_IF;
   IF #_w1 THEN
       "3号梯向上回一楼信号" := TRUE;
       "3号梯向下初始化信号" := FALSE;
   END_IF;
END_REGION

REGION Network 4: 平层信号
   RUNG wire#powerrail
      Contact( "3号梯向上回一楼信号" )
      Contact( "3号梯上平层信号" )
      Contact( "3号梯下平层信号" )
      wire#w1
      R_Coil( "3号梯上行接触器" )
   END_RUNG
   RUNG wire#w1
      R_Coil( "3号梯低速运行" )
   END_RUNG
   RUNG wire#w1
      S_Coil( "3号梯准备就绪信号" )
   END_RUNG
   RUNG wire#w1
      S_Coil( "3号梯风扇指示" )
   END_RUNG
   RUNG wire#w1
      S_Coil( "3号梯照明指示" )
   END_RUNG
   RUNG wire#w1
      R_Coil( "3号梯向上回一楼信号" )
   END_RUNG
   RUNG wire#w1
      Move(in := 1, out1 => "3号梯当前楼层数")
   END_RUNG
   // the same network as SCL:
   IF "3号梯向上回一楼信号" AND "3号梯上平层信号" AND "3号梯下平层信号" THEN
       "3号梯上行接触器" := FALSE;
       "3号梯低速运行" := FALSE;
       "3号梯准备就绪信号" := TRUE;
       "3号梯风扇指示" := TRUE;
       "3号梯照明指示" := TRUE;
   END_IF;
   #_w1 := "3号梯向上回一楼信号" AND "3号梯上平层信号" AND "3号梯下平层信号";
   IF #_w1 THEN
       "3号梯向上回一楼信号" := FALSE;
       "3号梯当前楼层数" := 1;
   END_IF;
END_REGION

REGION Network 5: 向上初始化
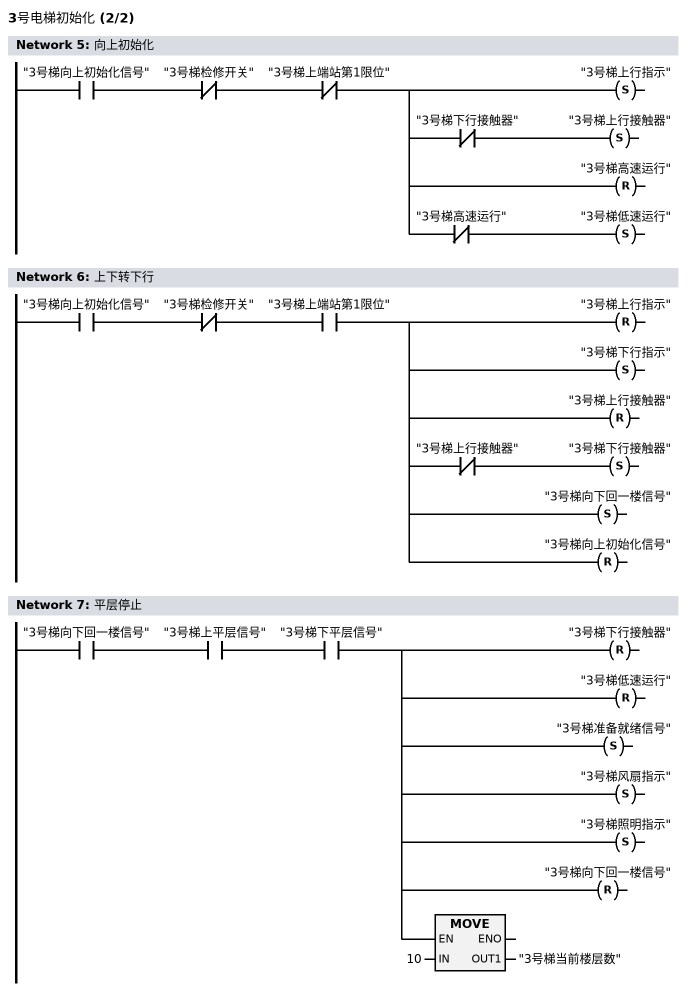
   RUNG wire#powerrail
      Contact( "3号梯向上初始化信号" )
      I_Contact( "3号梯检修开关" )
      I_Contact( "3号梯上端站第1限位" )
      wire#w1
      S_Coil( "3号梯上行指示" )
   END_RUNG
   RUNG wire#w1
      I_Contact( "3号梯下行接触器" )
      S_Coil( "3号梯上行接触器" )
   END_RUNG
   RUNG wire#w1
      R_Coil( "3号梯高速运行" )
   END_RUNG
   RUNG wire#w1
      I_Contact( "3号梯高速运行" )
      S_Coil( "3号梯低速运行" )
   END_RUNG
   // the same network as SCL:
   #_w1 := "3号梯向上初始化信号" AND NOT "3号梯检修开关" AND NOT "3号梯上端站第1限位";
   IF #_w1 THEN "3号梯上行指示" := TRUE; END_IF;
   IF #_w1 AND NOT "3号梯下行接触器" THEN "3号梯上行接触器" := TRUE; END_IF;
   IF #_w1 THEN "3号梯高速运行" := FALSE; END_IF;
   IF #_w1 AND NOT "3号梯高速运行" THEN "3号梯低速运行" := TRUE; END_IF;
END_REGION

REGION Network 6: 上下转下行
   RUNG wire#powerrail
      Contact( "3号梯向上初始化信号" )
      I_Contact( "3号梯检修开关" )
      Contact( "3号梯上端站第1限位" )
      wire#w1
      R_Coil( "3号梯上行指示" )
   END_RUNG
   RUNG wire#w1
      S_Coil( "3号梯下行指示" )
   END_RUNG
   RUNG wire#w1
      R_Coil( "3号梯上行接触器" )
   END_RUNG
   RUNG wire#w1
      I_Contact( "3号梯上行接触器" )
      S_Coil( "3号梯下行接触器" )
   END_RUNG
   RUNG wire#w1
      S_Coil( "3号梯向下回一楼信号" )
   END_RUNG
   RUNG wire#w1
      R_Coil( "3号梯向上初始化信号" )
   END_RUNG
   // the same network as SCL:
   #_w1 := "3号梯向上初始化信号" AND NOT "3号梯检修开关" AND "3号梯上端站第1限位";
   IF #_w1 THEN
       "3号梯上行指示" := FALSE;
       "3号梯下行指示" := TRUE;
       "3号梯上行接触器" := FALSE;
   END_IF;
   IF #_w1 AND NOT "3号梯上行接触器" THEN "3号梯下行接触器" := TRUE; END_IF;
   IF #_w1 THEN
       "3号梯向下回一楼信号" := TRUE;
       "3号梯向上初始化信号" := FALSE;
   END_IF;
END_REGION

REGION Network 7: 平层停止
   RUNG wire#powerrail
      Contact( "3号梯向下回一楼信号" )
      Contact( "3号梯上平层信号" )
      Contact( "3号梯下平层信号" )
      wire#w1
      R_Coil( "3号梯下行接触器" )
   END_RUNG
   RUNG wire#w1
      R_Coil( "3号梯低速运行" )
   END_RUNG
   RUNG wire#w1
      S_Coil( "3号梯准备就绪信号" )
   END_RUNG
   RUNG wire#w1
      S_Coil( "3号梯风扇指示" )
   END_RUNG
   RUNG wire#w1
      S_Coil( "3号梯照明指示" )
   END_RUNG
   RUNG wire#w1
      R_Coil( "3号梯向下回一楼信号" )
   END_RUNG
   RUNG wire#w1
      Move(in := 10, out1 => "3号梯当前楼层数")
   END_RUNG
   // the same network as SCL:
   IF "3号梯向下回一楼信号" AND "3号梯上平层信号" AND "3号梯下平层信号" THEN
       "3号梯下行接触器" := FALSE;
       "3号梯低速运行" := FALSE;
       "3号梯准备就绪信号" := TRUE;
       "3号梯风扇指示" := TRUE;
       "3号梯照明指示" := TRUE;
   END_IF;
   #_w1 := "3号梯向下回一楼信号" AND "3号梯上平层信号" AND "3号梯下平层信号";
   IF #_w1 THEN
       "3号梯向下回一楼信号" := FALSE;
       "3号梯当前楼层数" := 10;
   END_IF;
END_REGION
END_FUNCTION

FUNCTION "2号梯开门信号" : Void   // FC25, LAD
{ S7_Optimized_Access := 'TRUE' }
VERSION : 0.1
BEGIN

REGION Network 1: 本层开门
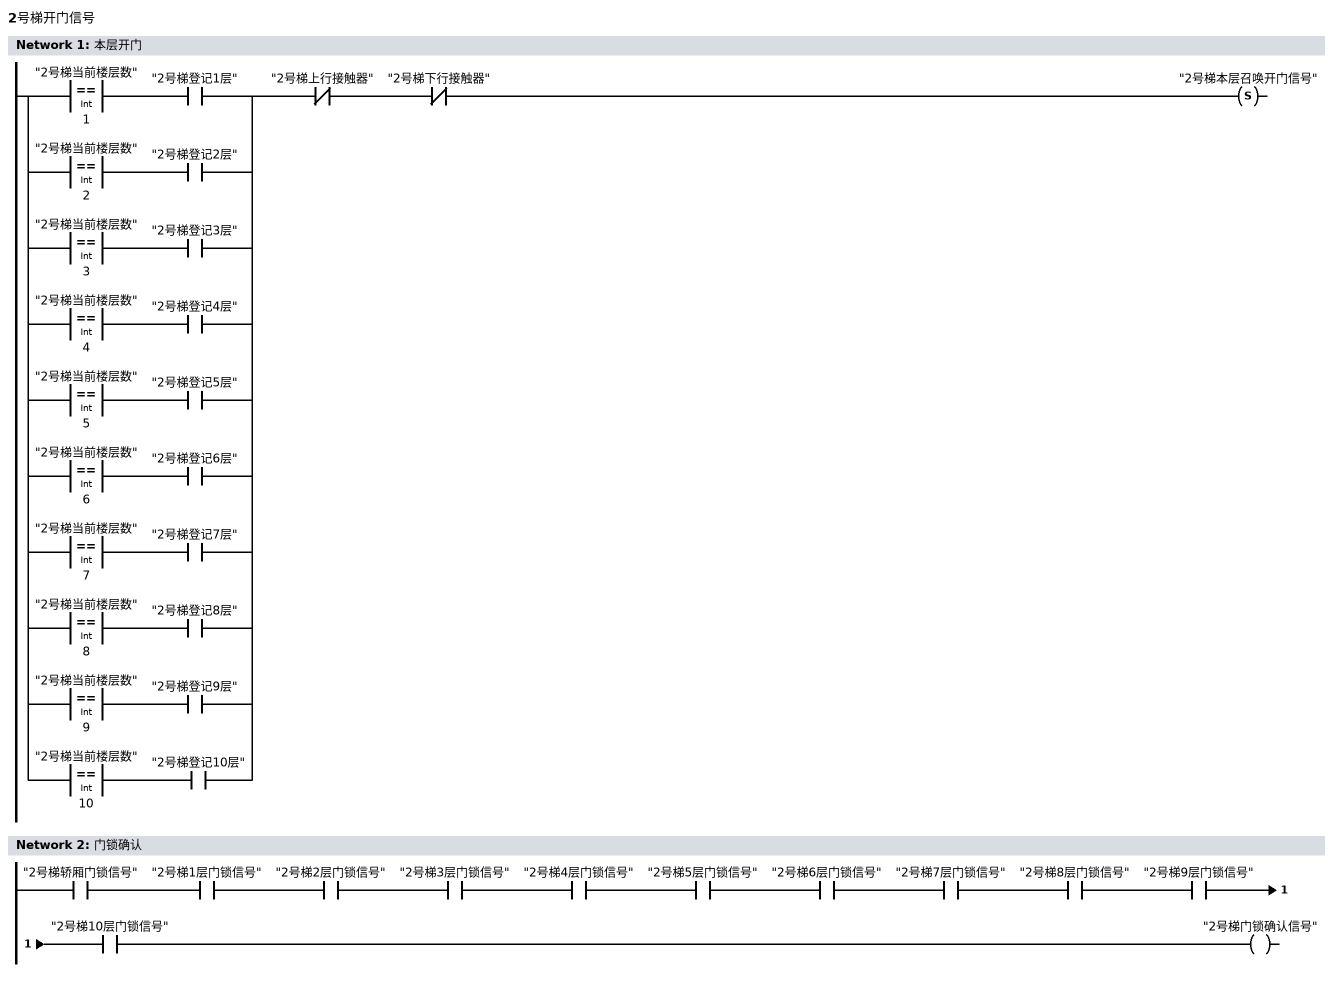
   RUNG wire#powerrail
      { S7_Templates := "SrcType := Int" } EQ_Contact(in1 := "2号梯当前楼层数", in2 := 1)
      Contact( "2号梯登记1层" )
      wire#w1
      I_Contact( "2号梯上行接触器" )
      I_Contact( "2号梯下行接触器" )
      S_Coil( "2号梯本层召唤开门信号" )
   END_RUNG
   RUNG wire#powerrail
      { S7_Templates := "SrcType := Int" } EQ_Contact(in1 := "2号梯当前楼层数", in2 := 2)
      Contact( "2号梯登记2层" )
   END_RUNG wire#w1
   RUNG wire#powerrail
      { S7_Templates := "SrcType := Int" } EQ_Contact(in1 := "2号梯当前楼层数", in2 := 3)
      Contact( "2号梯登记3层" )
   END_RUNG wire#w1
   RUNG wire#powerrail
      { S7_Templates := "SrcType := Int" } EQ_Contact(in1 := "2号梯当前楼层数", in2 := 4)
      Contact( "2号梯登记4层" )
   END_RUNG wire#w1
   RUNG wire#powerrail
      { S7_Templates := "SrcType := Int" } EQ_Contact(in1 := "2号梯当前楼层数", in2 := 5)
      Contact( "2号梯登记5层" )
   END_RUNG wire#w1
   RUNG wire#powerrail
      { S7_Templates := "SrcType := Int" } EQ_Contact(in1 := "2号梯当前楼层数", in2 := 6)
      Contact( "2号梯登记6层" )
   END_RUNG wire#w1
   RUNG wire#powerrail
      { S7_Templates := "SrcType := Int" } EQ_Contact(in1 := "2号梯当前楼层数", in2 := 7)
      Contact( "2号梯登记7层" )
   END_RUNG wire#w1
   RUNG wire#powerrail
      { S7_Templates := "SrcType := Int" } EQ_Contact(in1 := "2号梯当前楼层数", in2 := 8)
      Contact( "2号梯登记8层" )
   END_RUNG wire#w1
   RUNG wire#powerrail
      { S7_Templates := "SrcType := Int" } EQ_Contact(in1 := "2号梯当前楼层数", in2 := 9)
      Contact( "2号梯登记9层" )
   END_RUNG wire#w1
   RUNG wire#powerrail
      { S7_Templates := "SrcType := Int" } EQ_Contact(in1 := "2号梯当前楼层数", in2 := 10)
      Contact( "2号梯登记10层" )
   END_RUNG wire#w1
   // the same network as SCL:
   IF ((("2号梯当前楼层数" = 1) AND "2号梯登记1层") OR (("2号梯当前楼层数" = 2) AND "2号梯登记2层") OR (("2号梯当前楼层数" = 3) AND "2号梯登记3层") OR (("2号梯当前楼层数" = 4) AND "2号梯登记4层") OR (("2号梯当前楼层数" = 5) AND "2号梯登记5层") OR (("2号梯当前楼层数" = 6) AND "2号梯登记6层") OR (("2号梯当前楼层数" = 7) AND "2号梯登记7层") OR (("2号梯当前楼层数" = 8) AND "2号梯登记8层") OR (("2号梯当前楼层数" = 9) AND "2号梯登记9层") OR (("2号梯当前楼层数" = 10) AND "2号梯登记10层")) AND NOT "2号梯上行接触器" AND NOT "2号梯下行接触器" THEN
       "2号梯本层召唤开门信号" := TRUE;
   END_IF;
END_REGION

REGION Network 2: 门锁确认
   RUNG wire#powerrail
      Contact( "2号梯轿厢门锁信号" )
      Contact( "2号梯1层门锁信号" )
      Contact( "2号梯2层门锁信号" )
      Contact( "2号梯3层门锁信号" )
      Contact( "2号梯4层门锁信号" )
      Contact( "2号梯5层门锁信号" )
      Contact( "2号梯6层门锁信号" )
      Contact( "2号梯7层门锁信号" )
      Contact( "2号梯8层门锁信号" )
      Contact( "2号梯9层门锁信号" )
      Contact( "2号梯10层门锁信号" )
      Coil( "2号梯门锁确认信号" )
   END_RUNG
   // the same network as SCL:
   "2号梯门锁确认信号" := "2号梯轿厢门锁信号" AND "2号梯1层门锁信号" AND "2号梯2层门锁信号" AND "2号梯3层门锁信号" AND "2号梯4层门锁信号" AND "2号梯5层门锁信号" AND "2号梯6层门锁信号" AND "2号梯7层门锁信号" AND "2号梯8层门锁信号" AND "2号梯9层门锁信号" AND "2号梯10层门锁信号";
END_REGION
END_FUNCTION

FUNCTION "3号梯开门信号" : Void   // FC26, LAD
{ S7_Optimized_Access := 'TRUE' }
VERSION : 0.1
BEGIN

REGION Network 1: 本层开门
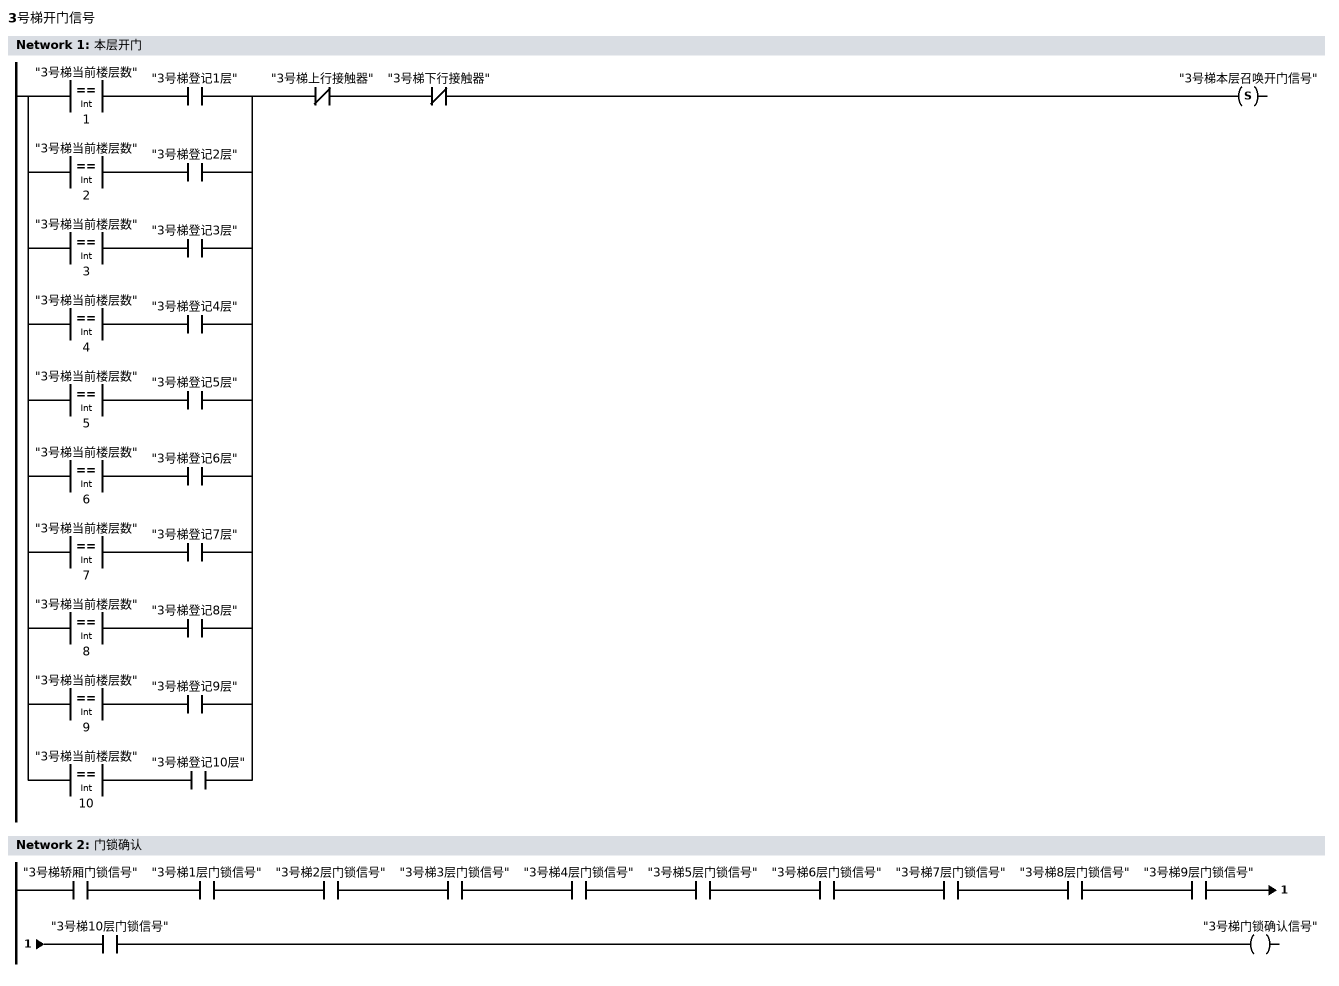
   RUNG wire#powerrail
      { S7_Templates := "SrcType := Int" } EQ_Contact(in1 := "3号梯当前楼层数", in2 := 1)
      Contact( "3号梯登记1层" )
      wire#w1
      I_Contact( "3号梯上行接触器" )
      I_Contact( "3号梯下行接触器" )
      S_Coil( "3号梯本层召唤开门信号" )
   END_RUNG
   RUNG wire#powerrail
      { S7_Templates := "SrcType := Int" } EQ_Contact(in1 := "3号梯当前楼层数", in2 := 2)
      Contact( "3号梯登记2层" )
   END_RUNG wire#w1
   RUNG wire#powerrail
      { S7_Templates := "SrcType := Int" } EQ_Contact(in1 := "3号梯当前楼层数", in2 := 3)
      Contact( "3号梯登记3层" )
   END_RUNG wire#w1
   RUNG wire#powerrail
      { S7_Templates := "SrcType := Int" } EQ_Contact(in1 := "3号梯当前楼层数", in2 := 4)
      Contact( "3号梯登记4层" )
   END_RUNG wire#w1
   RUNG wire#powerrail
      { S7_Templates := "SrcType := Int" } EQ_Contact(in1 := "3号梯当前楼层数", in2 := 5)
      Contact( "3号梯登记5层" )
   END_RUNG wire#w1
   RUNG wire#powerrail
      { S7_Templates := "SrcType := Int" } EQ_Contact(in1 := "3号梯当前楼层数", in2 := 6)
      Contact( "3号梯登记6层" )
   END_RUNG wire#w1
   RUNG wire#powerrail
      { S7_Templates := "SrcType := Int" } EQ_Contact(in1 := "3号梯当前楼层数", in2 := 7)
      Contact( "3号梯登记7层" )
   END_RUNG wire#w1
   RUNG wire#powerrail
      { S7_Templates := "SrcType := Int" } EQ_Contact(in1 := "3号梯当前楼层数", in2 := 8)
      Contact( "3号梯登记8层" )
   END_RUNG wire#w1
   RUNG wire#powerrail
      { S7_Templates := "SrcType := Int" } EQ_Contact(in1 := "3号梯当前楼层数", in2 := 9)
      Contact( "3号梯登记9层" )
   END_RUNG wire#w1
   RUNG wire#powerrail
      { S7_Templates := "SrcType := Int" } EQ_Contact(in1 := "3号梯当前楼层数", in2 := 10)
      Contact( "3号梯登记10层" )
   END_RUNG wire#w1
   // the same network as SCL:
   IF ((("3号梯当前楼层数" = 1) AND "3号梯登记1层") OR (("3号梯当前楼层数" = 2) AND "3号梯登记2层") OR (("3号梯当前楼层数" = 3) AND "3号梯登记3层") OR (("3号梯当前楼层数" = 4) AND "3号梯登记4层") OR (("3号梯当前楼层数" = 5) AND "3号梯登记5层") OR (("3号梯当前楼层数" = 6) AND "3号梯登记6层") OR (("3号梯当前楼层数" = 7) AND "3号梯登记7层") OR (("3号梯当前楼层数" = 8) AND "3号梯登记8层") OR (("3号梯当前楼层数" = 9) AND "3号梯登记9层") OR (("3号梯当前楼层数" = 10) AND "3号梯登记10层")) AND NOT "3号梯上行接触器" AND NOT "3号梯下行接触器" THEN
       "3号梯本层召唤开门信号" := TRUE;
   END_IF;
END_REGION

REGION Network 2: 门锁确认
   RUNG wire#powerrail
      Contact( "3号梯轿厢门锁信号" )
      Contact( "3号梯1层门锁信号" )
      Contact( "3号梯2层门锁信号" )
      Contact( "3号梯3层门锁信号" )
      Contact( "3号梯4层门锁信号" )
      Contact( "3号梯5层门锁信号" )
      Contact( "3号梯6层门锁信号" )
      Contact( "3号梯7层门锁信号" )
      Contact( "3号梯8层门锁信号" )
      Contact( "3号梯9层门锁信号" )
      Contact( "3号梯10层门锁信号" )
      Coil( "3号梯门锁确认信号" )
   END_RUNG
   // the same network as SCL:
   "3号梯门锁确认信号" := "3号梯轿厢门锁信号" AND "3号梯1层门锁信号" AND "3号梯2层门锁信号" AND "3号梯3层门锁信号" AND "3号梯4层门锁信号" AND "3号梯5层门锁信号" AND "3号梯6层门锁信号" AND "3号梯7层门锁信号" AND "3号梯8层门锁信号" AND "3号梯9层门锁信号" AND "3号梯10层门锁信号";
END_REGION
END_FUNCTION

FUNCTION "2号梯指示灯控制" : Void   // FC27, LAD
{ S7_Optimized_Access := 'TRUE' }
VERSION : 0.1
   VAR_TEMP   // added for the SCL form of the ladder/FBD networks
      _w1 : Bool;
      _w2 : Bool;
      _w3 : Bool;
      _w4 : Bool;
      _w5 : Bool;
      _w6 : Bool;
      _w7 : Bool;
      _w8 : Bool;
      _w9 : Bool;
   END_VAR
BEGIN

REGION Network 1: 2号梯终止下呼
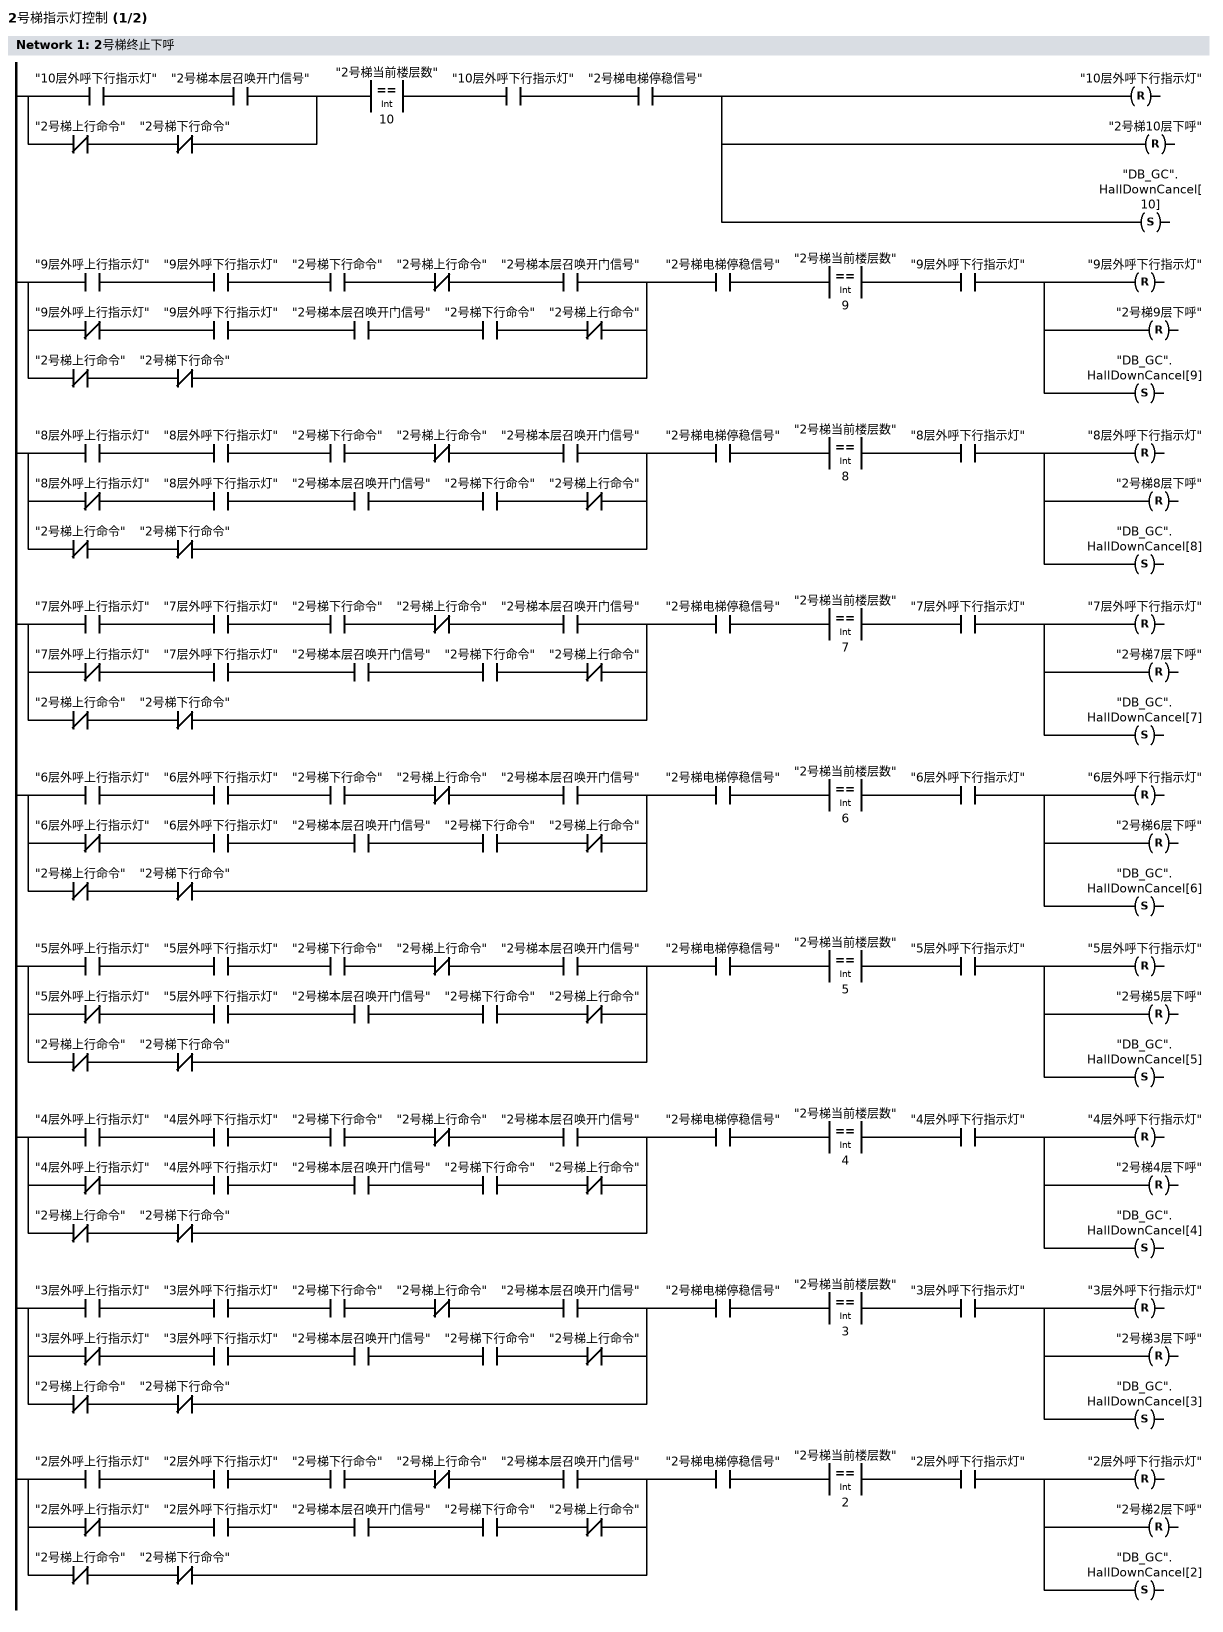
   RUNG wire#powerrail
      Contact( "10层外呼下行指示灯" )
      Contact( "2号梯本层召唤开门信号" )
      wire#w1
      { S7_Templates := "SrcType := Int" } EQ_Contact(in1 := "2号梯当前楼层数", in2 := 10)
      Contact( "10层外呼下行指示灯" )
      Contact( "2号梯电梯停稳信号" )
      wire#w2
      R_Coil( "10层外呼下行指示灯" )
   END_RUNG
   RUNG wire#powerrail
      I_Contact( "2号梯上行命令" )
      I_Contact( "2号梯下行命令" )
   END_RUNG wire#w1
   RUNG wire#w2
      R_Coil( "2号梯10层下呼" )
   END_RUNG
   RUNG wire#w2
      S_Coil( "DB_GC".HallDownCancel[10] )
   END_RUNG
   RUNG wire#powerrail
      Contact( "9层外呼上行指示灯" )
      Contact( "9层外呼下行指示灯" )
      Contact( "2号梯下行命令" )
      I_Contact( "2号梯上行命令" )
      Contact( "2号梯本层召唤开门信号" )
      wire#w3
      Contact( "2号梯电梯停稳信号" )
      { S7_Templates := "SrcType := Int" } EQ_Contact(in1 := "2号梯当前楼层数", in2 := 9)
      Contact( "9层外呼下行指示灯" )
      wire#w4
      R_Coil( "9层外呼下行指示灯" )
   END_RUNG
   RUNG wire#powerrail
      I_Contact( "9层外呼上行指示灯" )
      Contact( "9层外呼下行指示灯" )
      Contact( "2号梯本层召唤开门信号" )
      Contact( "2号梯下行命令" )
      I_Contact( "2号梯上行命令" )
   END_RUNG wire#w3
   RUNG wire#powerrail
      I_Contact( "2号梯上行命令" )
      I_Contact( "2号梯下行命令" )
   END_RUNG wire#w3
   RUNG wire#w4
      R_Coil( "2号梯9层下呼" )
   END_RUNG
   RUNG wire#w4
      S_Coil( "DB_GC".HallDownCancel[9] )
   END_RUNG
   RUNG wire#powerrail
      Contact( "8层外呼上行指示灯" )
      Contact( "8层外呼下行指示灯" )
      Contact( "2号梯下行命令" )
      I_Contact( "2号梯上行命令" )
      Contact( "2号梯本层召唤开门信号" )
      wire#w5
      Contact( "2号梯电梯停稳信号" )
      { S7_Templates := "SrcType := Int" } EQ_Contact(in1 := "2号梯当前楼层数", in2 := 8)
      Contact( "8层外呼下行指示灯" )
      wire#w6
      R_Coil( "8层外呼下行指示灯" )
   END_RUNG
   RUNG wire#powerrail
      I_Contact( "8层外呼上行指示灯" )
      Contact( "8层外呼下行指示灯" )
      Contact( "2号梯本层召唤开门信号" )
      Contact( "2号梯下行命令" )
      I_Contact( "2号梯上行命令" )
   END_RUNG wire#w5
   RUNG wire#powerrail
      I_Contact( "2号梯上行命令" )
      I_Contact( "2号梯下行命令" )
   END_RUNG wire#w5
   RUNG wire#w6
      R_Coil( "2号梯8层下呼" )
   END_RUNG
   RUNG wire#w6
      S_Coil( "DB_GC".HallDownCancel[8] )
   END_RUNG
   RUNG wire#powerrail
      Contact( "7层外呼上行指示灯" )
      Contact( "7层外呼下行指示灯" )
      Contact( "2号梯下行命令" )
      I_Contact( "2号梯上行命令" )
      Contact( "2号梯本层召唤开门信号" )
      wire#w7
      Contact( "2号梯电梯停稳信号" )
      { S7_Templates := "SrcType := Int" } EQ_Contact(in1 := "2号梯当前楼层数", in2 := 7)
      Contact( "7层外呼下行指示灯" )
      wire#w8
      R_Coil( "7层外呼下行指示灯" )
   END_RUNG
   RUNG wire#powerrail
      I_Contact( "7层外呼上行指示灯" )
      Contact( "7层外呼下行指示灯" )
      Contact( "2号梯本层召唤开门信号" )
      Contact( "2号梯下行命令" )
      I_Contact( "2号梯上行命令" )
   END_RUNG wire#w7
   RUNG wire#powerrail
      I_Contact( "2号梯上行命令" )
      I_Contact( "2号梯下行命令" )
   END_RUNG wire#w7
   RUNG wire#w8
      R_Coil( "2号梯7层下呼" )
   END_RUNG
   RUNG wire#w8
      S_Coil( "DB_GC".HallDownCancel[7] )
   END_RUNG
   RUNG wire#powerrail
      Contact( "6层外呼上行指示灯" )
      Contact( "6层外呼下行指示灯" )
      Contact( "2号梯下行命令" )
      I_Contact( "2号梯上行命令" )
      Contact( "2号梯本层召唤开门信号" )
      wire#w9
      Contact( "2号梯电梯停稳信号" )
      { S7_Templates := "SrcType := Int" } EQ_Contact(in1 := "2号梯当前楼层数", in2 := 6)
      Contact( "6层外呼下行指示灯" )
      wire#w10
      R_Coil( "6层外呼下行指示灯" )
   END_RUNG
   RUNG wire#powerrail
      I_Contact( "6层外呼上行指示灯" )
      Contact( "6层外呼下行指示灯" )
      Contact( "2号梯本层召唤开门信号" )
      Contact( "2号梯下行命令" )
      I_Contact( "2号梯上行命令" )
   END_RUNG wire#w9
   RUNG wire#powerrail
      I_Contact( "2号梯上行命令" )
      I_Contact( "2号梯下行命令" )
   END_RUNG wire#w9
   RUNG wire#w10
      R_Coil( "2号梯6层下呼" )
   END_RUNG
   RUNG wire#w10
      S_Coil( "DB_GC".HallDownCancel[6] )
   END_RUNG
   RUNG wire#powerrail
      Contact( "5层外呼上行指示灯" )
      Contact( "5层外呼下行指示灯" )
      Contact( "2号梯下行命令" )
      I_Contact( "2号梯上行命令" )
      Contact( "2号梯本层召唤开门信号" )
      wire#w11
      Contact( "2号梯电梯停稳信号" )
      { S7_Templates := "SrcType := Int" } EQ_Contact(in1 := "2号梯当前楼层数", in2 := 5)
      Contact( "5层外呼下行指示灯" )
      wire#w12
      R_Coil( "5层外呼下行指示灯" )
   END_RUNG
   RUNG wire#powerrail
      I_Contact( "5层外呼上行指示灯" )
      Contact( "5层外呼下行指示灯" )
      Contact( "2号梯本层召唤开门信号" )
      Contact( "2号梯下行命令" )
      I_Contact( "2号梯上行命令" )
   END_RUNG wire#w11
   RUNG wire#powerrail
      I_Contact( "2号梯上行命令" )
      I_Contact( "2号梯下行命令" )
   END_RUNG wire#w11
   RUNG wire#w12
      R_Coil( "2号梯5层下呼" )
   END_RUNG
   RUNG wire#w12
      S_Coil( "DB_GC".HallDownCancel[5] )
   END_RUNG
   RUNG wire#powerrail
      Contact( "4层外呼上行指示灯" )
      Contact( "4层外呼下行指示灯" )
      Contact( "2号梯下行命令" )
      I_Contact( "2号梯上行命令" )
      Contact( "2号梯本层召唤开门信号" )
      wire#w13
      Contact( "2号梯电梯停稳信号" )
      { S7_Templates := "SrcType := Int" } EQ_Contact(in1 := "2号梯当前楼层数", in2 := 4)
      Contact( "4层外呼下行指示灯" )
      wire#w14
      R_Coil( "4层外呼下行指示灯" )
   END_RUNG
   RUNG wire#powerrail
      I_Contact( "4层外呼上行指示灯" )
      Contact( "4层外呼下行指示灯" )
      Contact( "2号梯本层召唤开门信号" )
      Contact( "2号梯下行命令" )
      I_Contact( "2号梯上行命令" )
   END_RUNG wire#w13
   RUNG wire#powerrail
      I_Contact( "2号梯上行命令" )
      I_Contact( "2号梯下行命令" )
   END_RUNG wire#w13
   RUNG wire#w14
      R_Coil( "2号梯4层下呼" )
   END_RUNG
   RUNG wire#w14
      S_Coil( "DB_GC".HallDownCancel[4] )
   END_RUNG
   RUNG wire#powerrail
      Contact( "3层外呼上行指示灯" )
      Contact( "3层外呼下行指示灯" )
      Contact( "2号梯下行命令" )
      I_Contact( "2号梯上行命令" )
      Contact( "2号梯本层召唤开门信号" )
      wire#w15
      Contact( "2号梯电梯停稳信号" )
      { S7_Templates := "SrcType := Int" } EQ_Contact(in1 := "2号梯当前楼层数", in2 := 3)
      Contact( "3层外呼下行指示灯" )
      wire#w16
      R_Coil( "3层外呼下行指示灯" )
   END_RUNG
   RUNG wire#powerrail
      I_Contact( "3层外呼上行指示灯" )
      Contact( "3层外呼下行指示灯" )
      Contact( "2号梯本层召唤开门信号" )
      Contact( "2号梯下行命令" )
      I_Contact( "2号梯上行命令" )
   END_RUNG wire#w15
   RUNG wire#powerrail
      I_Contact( "2号梯上行命令" )
      I_Contact( "2号梯下行命令" )
   END_RUNG wire#w15
   RUNG wire#w16
      R_Coil( "2号梯3层下呼" )
   END_RUNG
   RUNG wire#w16
      S_Coil( "DB_GC".HallDownCancel[3] )
   END_RUNG
   RUNG wire#powerrail
      Contact( "2层外呼上行指示灯" )
      Contact( "2层外呼下行指示灯" )
      Contact( "2号梯下行命令" )
      I_Contact( "2号梯上行命令" )
      Contact( "2号梯本层召唤开门信号" )
      wire#w17
      Contact( "2号梯电梯停稳信号" )
      { S7_Templates := "SrcType := Int" } EQ_Contact(in1 := "2号梯当前楼层数", in2 := 2)
      Contact( "2层外呼下行指示灯" )
      wire#w18
      R_Coil( "2层外呼下行指示灯" )
   END_RUNG
   RUNG wire#powerrail
      I_Contact( "2层外呼上行指示灯" )
      Contact( "2层外呼下行指示灯" )
      Contact( "2号梯本层召唤开门信号" )
      Contact( "2号梯下行命令" )
      I_Contact( "2号梯上行命令" )
   END_RUNG wire#w17
   RUNG wire#powerrail
      I_Contact( "2号梯上行命令" )
      I_Contact( "2号梯下行命令" )
   END_RUNG wire#w17
   RUNG wire#w18
      R_Coil( "2号梯2层下呼" )
   END_RUNG
   RUNG wire#w18
      S_Coil( "DB_GC".HallDownCancel[2] )
   END_RUNG
   // the same network as SCL:
   #_w1 := (("10层外呼下行指示灯" AND "2号梯本层召唤开门信号") OR (NOT "2号梯上行命令" AND NOT "2号梯下行命令")) AND ("2号梯当前楼层数" = 10) AND "10层外呼下行指示灯" AND "2号梯电梯停稳信号";
   IF #_w1 THEN
       "10层外呼下行指示灯" := FALSE;
       "2号梯10层下呼" := FALSE;
       "DB_GC".HallDownCancel[10] := TRUE;
   END_IF;
   #_w2 := (("9层外呼上行指示灯" AND "9层外呼下行指示灯" AND "2号梯下行命令" AND NOT "2号梯上行命令" AND "2号梯本层召唤开门信号") OR (NOT "9层外呼上行指示灯" AND "9层外呼下行指示灯" AND "2号梯本层召唤开门信号" AND "2号梯下行命令" AND NOT "2号梯上行命令") OR (NOT "2号梯上行命令" AND NOT "2号梯下行命令")) AND "2号梯电梯停稳信号" AND ("2号梯当前楼层数" = 9) AND "9层外呼下行指示灯";
   IF #_w2 THEN
       "9层外呼下行指示灯" := FALSE;
       "2号梯9层下呼" := FALSE;
       "DB_GC".HallDownCancel[9] := TRUE;
   END_IF;
   #_w3 := (("8层外呼上行指示灯" AND "8层外呼下行指示灯" AND "2号梯下行命令" AND NOT "2号梯上行命令" AND "2号梯本层召唤开门信号") OR (NOT "8层外呼上行指示灯" AND "8层外呼下行指示灯" AND "2号梯本层召唤开门信号" AND "2号梯下行命令" AND NOT "2号梯上行命令") OR (NOT "2号梯上行命令" AND NOT "2号梯下行命令")) AND "2号梯电梯停稳信号" AND ("2号梯当前楼层数" = 8) AND "8层外呼下行指示灯";
   IF #_w3 THEN
       "8层外呼下行指示灯" := FALSE;
       "2号梯8层下呼" := FALSE;
       "DB_GC".HallDownCancel[8] := TRUE;
   END_IF;
   #_w4 := (("7层外呼上行指示灯" AND "7层外呼下行指示灯" AND "2号梯下行命令" AND NOT "2号梯上行命令" AND "2号梯本层召唤开门信号") OR (NOT "7层外呼上行指示灯" AND "7层外呼下行指示灯" AND "2号梯本层召唤开门信号" AND "2号梯下行命令" AND NOT "2号梯上行命令") OR (NOT "2号梯上行命令" AND NOT "2号梯下行命令")) AND "2号梯电梯停稳信号" AND ("2号梯当前楼层数" = 7) AND "7层外呼下行指示灯";
   IF #_w4 THEN
       "7层外呼下行指示灯" := FALSE;
       "2号梯7层下呼" := FALSE;
       "DB_GC".HallDownCancel[7] := TRUE;
   END_IF;
   #_w5 := (("6层外呼上行指示灯" AND "6层外呼下行指示灯" AND "2号梯下行命令" AND NOT "2号梯上行命令" AND "2号梯本层召唤开门信号") OR (NOT "6层外呼上行指示灯" AND "6层外呼下行指示灯" AND "2号梯本层召唤开门信号" AND "2号梯下行命令" AND NOT "2号梯上行命令") OR (NOT "2号梯上行命令" AND NOT "2号梯下行命令")) AND "2号梯电梯停稳信号" AND ("2号梯当前楼层数" = 6) AND "6层外呼下行指示灯";
   IF #_w5 THEN
       "6层外呼下行指示灯" := FALSE;
       "2号梯6层下呼" := FALSE;
       "DB_GC".HallDownCancel[6] := TRUE;
   END_IF;
   #_w6 := (("5层外呼上行指示灯" AND "5层外呼下行指示灯" AND "2号梯下行命令" AND NOT "2号梯上行命令" AND "2号梯本层召唤开门信号") OR (NOT "5层外呼上行指示灯" AND "5层外呼下行指示灯" AND "2号梯本层召唤开门信号" AND "2号梯下行命令" AND NOT "2号梯上行命令") OR (NOT "2号梯上行命令" AND NOT "2号梯下行命令")) AND "2号梯电梯停稳信号" AND ("2号梯当前楼层数" = 5) AND "5层外呼下行指示灯";
   IF #_w6 THEN
       "5层外呼下行指示灯" := FALSE;
       "2号梯5层下呼" := FALSE;
       "DB_GC".HallDownCancel[5] := TRUE;
   END_IF;
   #_w7 := (("4层外呼上行指示灯" AND "4层外呼下行指示灯" AND "2号梯下行命令" AND NOT "2号梯上行命令" AND "2号梯本层召唤开门信号") OR (NOT "4层外呼上行指示灯" AND "4层外呼下行指示灯" AND "2号梯本层召唤开门信号" AND "2号梯下行命令" AND NOT "2号梯上行命令") OR (NOT "2号梯上行命令" AND NOT "2号梯下行命令")) AND "2号梯电梯停稳信号" AND ("2号梯当前楼层数" = 4) AND "4层外呼下行指示灯";
   IF #_w7 THEN
       "4层外呼下行指示灯" := FALSE;
       "2号梯4层下呼" := FALSE;
       "DB_GC".HallDownCancel[4] := TRUE;
   END_IF;
   #_w8 := (("3层外呼上行指示灯" AND "3层外呼下行指示灯" AND "2号梯下行命令" AND NOT "2号梯上行命令" AND "2号梯本层召唤开门信号") OR (NOT "3层外呼上行指示灯" AND "3层外呼下行指示灯" AND "2号梯本层召唤开门信号" AND "2号梯下行命令" AND NOT "2号梯上行命令") OR (NOT "2号梯上行命令" AND NOT "2号梯下行命令")) AND "2号梯电梯停稳信号" AND ("2号梯当前楼层数" = 3) AND "3层外呼下行指示灯";
   IF #_w8 THEN
       "3层外呼下行指示灯" := FALSE;
       "2号梯3层下呼" := FALSE;
       "DB_GC".HallDownCancel[3] := TRUE;
   END_IF;
   #_w9 := (("2层外呼上行指示灯" AND "2层外呼下行指示灯" AND "2号梯下行命令" AND NOT "2号梯上行命令" AND "2号梯本层召唤开门信号") OR (NOT "2层外呼上行指示灯" AND "2层外呼下行指示灯" AND "2号梯本层召唤开门信号" AND "2号梯下行命令" AND NOT "2号梯上行命令") OR (NOT "2号梯上行命令" AND NOT "2号梯下行命令")) AND "2号梯电梯停稳信号" AND ("2号梯当前楼层数" = 2) AND "2层外呼下行指示灯";
   IF #_w9 THEN
       "2层外呼下行指示灯" := FALSE;
       "2号梯2层下呼" := FALSE;
       "DB_GC".HallDownCancel[2] := TRUE;
   END_IF;
END_REGION

REGION Network 2: 2号梯终止上呼
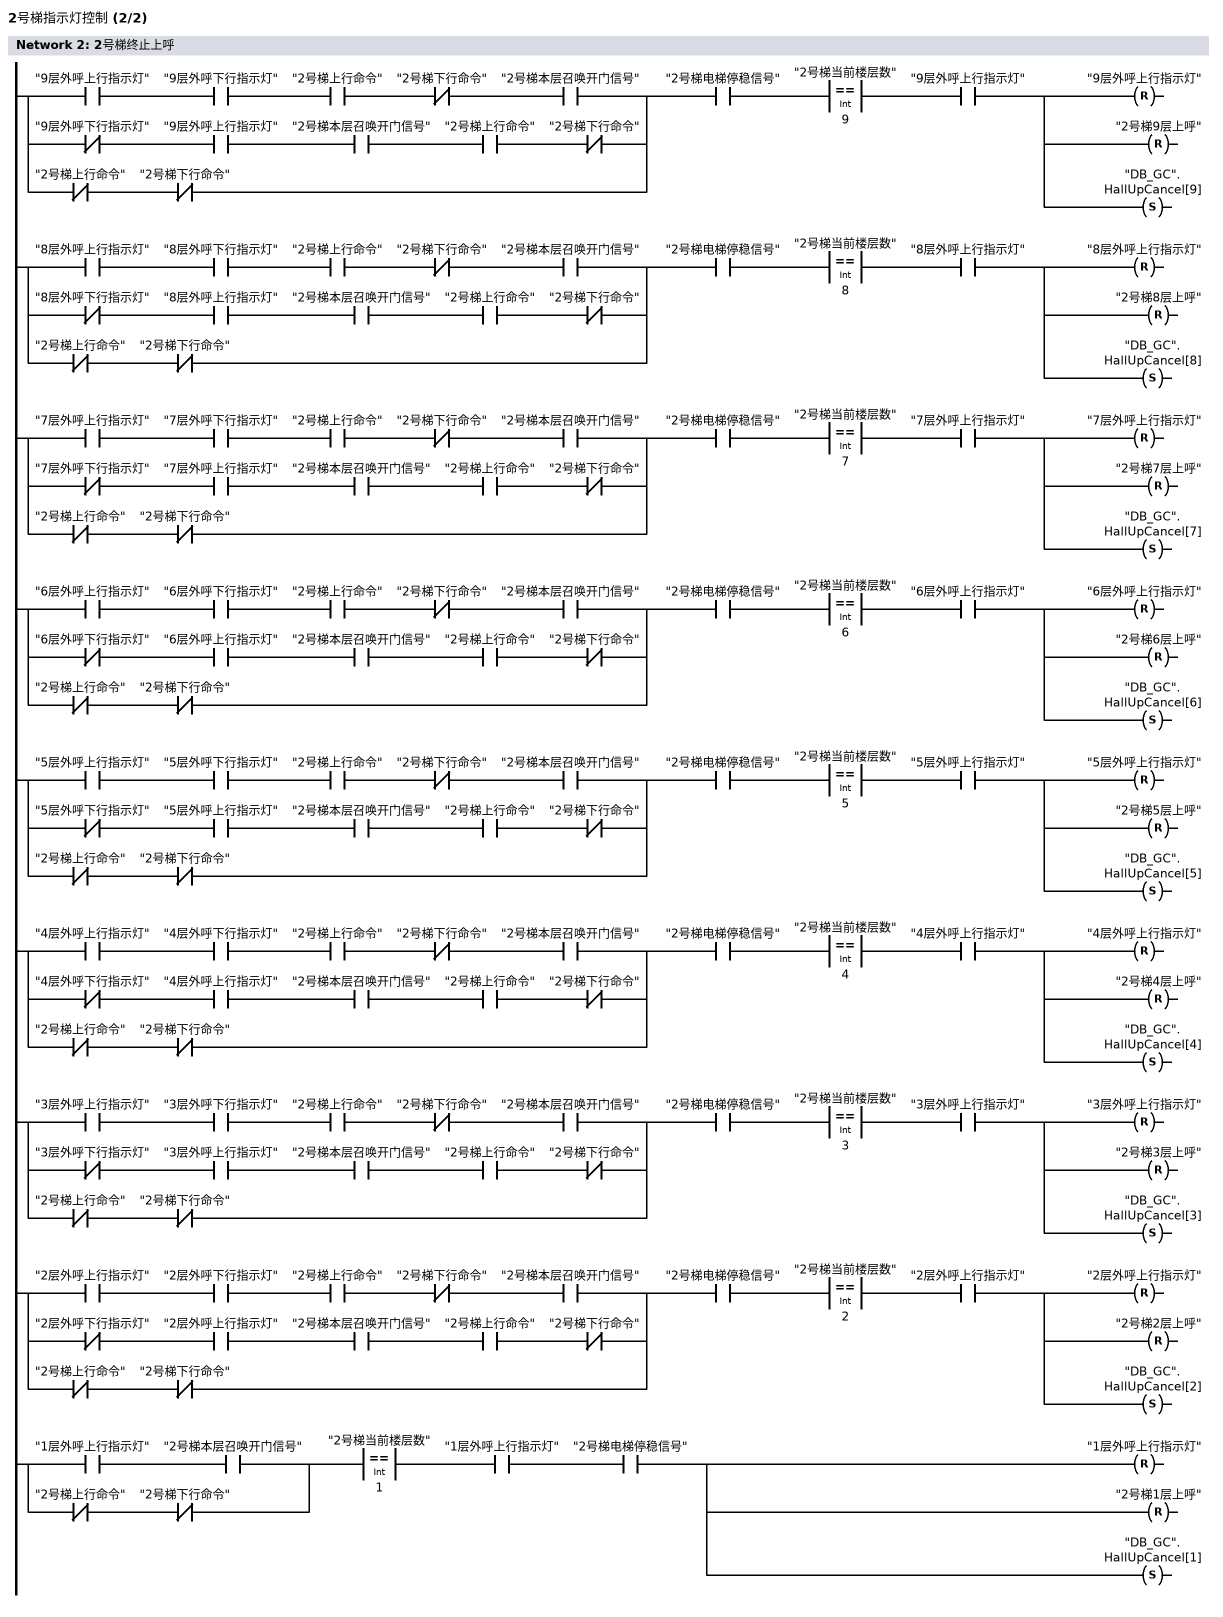
   RUNG wire#powerrail
      Contact( "9层外呼上行指示灯" )
      Contact( "9层外呼下行指示灯" )
      Contact( "2号梯上行命令" )
      I_Contact( "2号梯下行命令" )
      Contact( "2号梯本层召唤开门信号" )
      wire#w1
      Contact( "2号梯电梯停稳信号" )
      { S7_Templates := "SrcType := Int" } EQ_Contact(in1 := "2号梯当前楼层数", in2 := 9)
      Contact( "9层外呼上行指示灯" )
      wire#w2
      R_Coil( "9层外呼上行指示灯" )
   END_RUNG
   RUNG wire#powerrail
      I_Contact( "9层外呼下行指示灯" )
      Contact( "9层外呼上行指示灯" )
      Contact( "2号梯本层召唤开门信号" )
      Contact( "2号梯上行命令" )
      I_Contact( "2号梯下行命令" )
   END_RUNG wire#w1
   RUNG wire#powerrail
      I_Contact( "2号梯上行命令" )
      I_Contact( "2号梯下行命令" )
   END_RUNG wire#w1
   RUNG wire#w2
      R_Coil( "2号梯9层上呼" )
   END_RUNG
   RUNG wire#w2
      S_Coil( "DB_GC".HallUpCancel[9] )
   END_RUNG
   RUNG wire#powerrail
      Contact( "8层外呼上行指示灯" )
      Contact( "8层外呼下行指示灯" )
      Contact( "2号梯上行命令" )
      I_Contact( "2号梯下行命令" )
      Contact( "2号梯本层召唤开门信号" )
      wire#w3
      Contact( "2号梯电梯停稳信号" )
      { S7_Templates := "SrcType := Int" } EQ_Contact(in1 := "2号梯当前楼层数", in2 := 8)
      Contact( "8层外呼上行指示灯" )
      wire#w4
      R_Coil( "8层外呼上行指示灯" )
   END_RUNG
   RUNG wire#powerrail
      I_Contact( "8层外呼下行指示灯" )
      Contact( "8层外呼上行指示灯" )
      Contact( "2号梯本层召唤开门信号" )
      Contact( "2号梯上行命令" )
      I_Contact( "2号梯下行命令" )
   END_RUNG wire#w3
   RUNG wire#powerrail
      I_Contact( "2号梯上行命令" )
      I_Contact( "2号梯下行命令" )
   END_RUNG wire#w3
   RUNG wire#w4
      R_Coil( "2号梯8层上呼" )
   END_RUNG
   RUNG wire#w4
      S_Coil( "DB_GC".HallUpCancel[8] )
   END_RUNG
   RUNG wire#powerrail
      Contact( "7层外呼上行指示灯" )
      Contact( "7层外呼下行指示灯" )
      Contact( "2号梯上行命令" )
      I_Contact( "2号梯下行命令" )
      Contact( "2号梯本层召唤开门信号" )
      wire#w5
      Contact( "2号梯电梯停稳信号" )
      { S7_Templates := "SrcType := Int" } EQ_Contact(in1 := "2号梯当前楼层数", in2 := 7)
      Contact( "7层外呼上行指示灯" )
      wire#w6
      R_Coil( "7层外呼上行指示灯" )
   END_RUNG
   RUNG wire#powerrail
      I_Contact( "7层外呼下行指示灯" )
      Contact( "7层外呼上行指示灯" )
      Contact( "2号梯本层召唤开门信号" )
      Contact( "2号梯上行命令" )
      I_Contact( "2号梯下行命令" )
   END_RUNG wire#w5
   RUNG wire#powerrail
      I_Contact( "2号梯上行命令" )
      I_Contact( "2号梯下行命令" )
   END_RUNG wire#w5
   RUNG wire#w6
      R_Coil( "2号梯7层上呼" )
   END_RUNG
   RUNG wire#w6
      S_Coil( "DB_GC".HallUpCancel[7] )
   END_RUNG
   RUNG wire#powerrail
      Contact( "6层外呼上行指示灯" )
      Contact( "6层外呼下行指示灯" )
      Contact( "2号梯上行命令" )
      I_Contact( "2号梯下行命令" )
      Contact( "2号梯本层召唤开门信号" )
      wire#w7
      Contact( "2号梯电梯停稳信号" )
      { S7_Templates := "SrcType := Int" } EQ_Contact(in1 := "2号梯当前楼层数", in2 := 6)
      Contact( "6层外呼上行指示灯" )
      wire#w8
      R_Coil( "6层外呼上行指示灯" )
   END_RUNG
   RUNG wire#powerrail
      I_Contact( "6层外呼下行指示灯" )
      Contact( "6层外呼上行指示灯" )
      Contact( "2号梯本层召唤开门信号" )
      Contact( "2号梯上行命令" )
      I_Contact( "2号梯下行命令" )
   END_RUNG wire#w7
   RUNG wire#powerrail
      I_Contact( "2号梯上行命令" )
      I_Contact( "2号梯下行命令" )
   END_RUNG wire#w7
   RUNG wire#w8
      R_Coil( "2号梯6层上呼" )
   END_RUNG
   RUNG wire#w8
      S_Coil( "DB_GC".HallUpCancel[6] )
   END_RUNG
   RUNG wire#powerrail
      Contact( "5层外呼上行指示灯" )
      Contact( "5层外呼下行指示灯" )
      Contact( "2号梯上行命令" )
      I_Contact( "2号梯下行命令" )
      Contact( "2号梯本层召唤开门信号" )
      wire#w9
      Contact( "2号梯电梯停稳信号" )
      { S7_Templates := "SrcType := Int" } EQ_Contact(in1 := "2号梯当前楼层数", in2 := 5)
      Contact( "5层外呼上行指示灯" )
      wire#w10
      R_Coil( "5层外呼上行指示灯" )
   END_RUNG
   RUNG wire#powerrail
      I_Contact( "5层外呼下行指示灯" )
      Contact( "5层外呼上行指示灯" )
      Contact( "2号梯本层召唤开门信号" )
      Contact( "2号梯上行命令" )
      I_Contact( "2号梯下行命令" )
   END_RUNG wire#w9
   RUNG wire#powerrail
      I_Contact( "2号梯上行命令" )
      I_Contact( "2号梯下行命令" )
   END_RUNG wire#w9
   RUNG wire#w10
      R_Coil( "2号梯5层上呼" )
   END_RUNG
   RUNG wire#w10
      S_Coil( "DB_GC".HallUpCancel[5] )
   END_RUNG
   RUNG wire#powerrail
      Contact( "4层外呼上行指示灯" )
      Contact( "4层外呼下行指示灯" )
      Contact( "2号梯上行命令" )
      I_Contact( "2号梯下行命令" )
      Contact( "2号梯本层召唤开门信号" )
      wire#w11
      Contact( "2号梯电梯停稳信号" )
      { S7_Templates := "SrcType := Int" } EQ_Contact(in1 := "2号梯当前楼层数", in2 := 4)
      Contact( "4层外呼上行指示灯" )
      wire#w12
      R_Coil( "4层外呼上行指示灯" )
   END_RUNG
   RUNG wire#powerrail
      I_Contact( "4层外呼下行指示灯" )
      Contact( "4层外呼上行指示灯" )
      Contact( "2号梯本层召唤开门信号" )
      Contact( "2号梯上行命令" )
      I_Contact( "2号梯下行命令" )
   END_RUNG wire#w11
   RUNG wire#powerrail
      I_Contact( "2号梯上行命令" )
      I_Contact( "2号梯下行命令" )
   END_RUNG wire#w11
   RUNG wire#w12
      R_Coil( "2号梯4层上呼" )
   END_RUNG
   RUNG wire#w12
      S_Coil( "DB_GC".HallUpCancel[4] )
   END_RUNG
   RUNG wire#powerrail
      Contact( "3层外呼上行指示灯" )
      Contact( "3层外呼下行指示灯" )
      Contact( "2号梯上行命令" )
      I_Contact( "2号梯下行命令" )
      Contact( "2号梯本层召唤开门信号" )
      wire#w13
      Contact( "2号梯电梯停稳信号" )
      { S7_Templates := "SrcType := Int" } EQ_Contact(in1 := "2号梯当前楼层数", in2 := 3)
      Contact( "3层外呼上行指示灯" )
      wire#w14
      R_Coil( "3层外呼上行指示灯" )
   END_RUNG
   RUNG wire#powerrail
      I_Contact( "3层外呼下行指示灯" )
      Contact( "3层外呼上行指示灯" )
      Contact( "2号梯本层召唤开门信号" )
      Contact( "2号梯上行命令" )
      I_Contact( "2号梯下行命令" )
   END_RUNG wire#w13
   RUNG wire#powerrail
      I_Contact( "2号梯上行命令" )
      I_Contact( "2号梯下行命令" )
   END_RUNG wire#w13
   RUNG wire#w14
      R_Coil( "2号梯3层上呼" )
   END_RUNG
   RUNG wire#w14
      S_Coil( "DB_GC".HallUpCancel[3] )
   END_RUNG
   RUNG wire#powerrail
      Contact( "2层外呼上行指示灯" )
      Contact( "2层外呼下行指示灯" )
      Contact( "2号梯上行命令" )
      I_Contact( "2号梯下行命令" )
      Contact( "2号梯本层召唤开门信号" )
      wire#w15
      Contact( "2号梯电梯停稳信号" )
      { S7_Templates := "SrcType := Int" } EQ_Contact(in1 := "2号梯当前楼层数", in2 := 2)
      Contact( "2层外呼上行指示灯" )
      wire#w16
      R_Coil( "2层外呼上行指示灯" )
   END_RUNG
   RUNG wire#powerrail
      I_Contact( "2层外呼下行指示灯" )
      Contact( "2层外呼上行指示灯" )
      Contact( "2号梯本层召唤开门信号" )
      Contact( "2号梯上行命令" )
      I_Contact( "2号梯下行命令" )
   END_RUNG wire#w15
   RUNG wire#powerrail
      I_Contact( "2号梯上行命令" )
      I_Contact( "2号梯下行命令" )
   END_RUNG wire#w15
   RUNG wire#w16
      R_Coil( "2号梯2层上呼" )
   END_RUNG
   RUNG wire#w16
      S_Coil( "DB_GC".HallUpCancel[2] )
   END_RUNG
   RUNG wire#powerrail
      Contact( "1层外呼上行指示灯" )
      Contact( "2号梯本层召唤开门信号" )
      wire#w17
      { S7_Templates := "SrcType := Int" } EQ_Contact(in1 := "2号梯当前楼层数", in2 := 1)
      Contact( "1层外呼上行指示灯" )
      Contact( "2号梯电梯停稳信号" )
      wire#w18
      R_Coil( "1层外呼上行指示灯" )
   END_RUNG
   RUNG wire#powerrail
      I_Contact( "2号梯上行命令" )
      I_Contact( "2号梯下行命令" )
   END_RUNG wire#w17
   RUNG wire#w18
      R_Coil( "2号梯1层上呼" )
   END_RUNG
   RUNG wire#w18
      S_Coil( "DB_GC".HallUpCancel[1] )
   END_RUNG
   // the same network as SCL:
   #_w1 := (("9层外呼上行指示灯" AND "9层外呼下行指示灯" AND "2号梯上行命令" AND NOT "2号梯下行命令" AND "2号梯本层召唤开门信号") OR (NOT "9层外呼下行指示灯" AND "9层外呼上行指示灯" AND "2号梯本层召唤开门信号" AND "2号梯上行命令" AND NOT "2号梯下行命令") OR (NOT "2号梯上行命令" AND NOT "2号梯下行命令")) AND "2号梯电梯停稳信号" AND ("2号梯当前楼层数" = 9) AND "9层外呼上行指示灯";
   IF #_w1 THEN
       "9层外呼上行指示灯" := FALSE;
       "2号梯9层上呼" := FALSE;
       "DB_GC".HallUpCancel[9] := TRUE;
   END_IF;
   #_w2 := (("8层外呼上行指示灯" AND "8层外呼下行指示灯" AND "2号梯上行命令" AND NOT "2号梯下行命令" AND "2号梯本层召唤开门信号") OR (NOT "8层外呼下行指示灯" AND "8层外呼上行指示灯" AND "2号梯本层召唤开门信号" AND "2号梯上行命令" AND NOT "2号梯下行命令") OR (NOT "2号梯上行命令" AND NOT "2号梯下行命令")) AND "2号梯电梯停稳信号" AND ("2号梯当前楼层数" = 8) AND "8层外呼上行指示灯";
   IF #_w2 THEN
       "8层外呼上行指示灯" := FALSE;
       "2号梯8层上呼" := FALSE;
       "DB_GC".HallUpCancel[8] := TRUE;
   END_IF;
   #_w3 := (("7层外呼上行指示灯" AND "7层外呼下行指示灯" AND "2号梯上行命令" AND NOT "2号梯下行命令" AND "2号梯本层召唤开门信号") OR (NOT "7层外呼下行指示灯" AND "7层外呼上行指示灯" AND "2号梯本层召唤开门信号" AND "2号梯上行命令" AND NOT "2号梯下行命令") OR (NOT "2号梯上行命令" AND NOT "2号梯下行命令")) AND "2号梯电梯停稳信号" AND ("2号梯当前楼层数" = 7) AND "7层外呼上行指示灯";
   IF #_w3 THEN
       "7层外呼上行指示灯" := FALSE;
       "2号梯7层上呼" := FALSE;
       "DB_GC".HallUpCancel[7] := TRUE;
   END_IF;
   #_w4 := (("6层外呼上行指示灯" AND "6层外呼下行指示灯" AND "2号梯上行命令" AND NOT "2号梯下行命令" AND "2号梯本层召唤开门信号") OR (NOT "6层外呼下行指示灯" AND "6层外呼上行指示灯" AND "2号梯本层召唤开门信号" AND "2号梯上行命令" AND NOT "2号梯下行命令") OR (NOT "2号梯上行命令" AND NOT "2号梯下行命令")) AND "2号梯电梯停稳信号" AND ("2号梯当前楼层数" = 6) AND "6层外呼上行指示灯";
   IF #_w4 THEN
       "6层外呼上行指示灯" := FALSE;
       "2号梯6层上呼" := FALSE;
       "DB_GC".HallUpCancel[6] := TRUE;
   END_IF;
   #_w5 := (("5层外呼上行指示灯" AND "5层外呼下行指示灯" AND "2号梯上行命令" AND NOT "2号梯下行命令" AND "2号梯本层召唤开门信号") OR (NOT "5层外呼下行指示灯" AND "5层外呼上行指示灯" AND "2号梯本层召唤开门信号" AND "2号梯上行命令" AND NOT "2号梯下行命令") OR (NOT "2号梯上行命令" AND NOT "2号梯下行命令")) AND "2号梯电梯停稳信号" AND ("2号梯当前楼层数" = 5) AND "5层外呼上行指示灯";
   IF #_w5 THEN
       "5层外呼上行指示灯" := FALSE;
       "2号梯5层上呼" := FALSE;
       "DB_GC".HallUpCancel[5] := TRUE;
   END_IF;
   #_w6 := (("4层外呼上行指示灯" AND "4层外呼下行指示灯" AND "2号梯上行命令" AND NOT "2号梯下行命令" AND "2号梯本层召唤开门信号") OR (NOT "4层外呼下行指示灯" AND "4层外呼上行指示灯" AND "2号梯本层召唤开门信号" AND "2号梯上行命令" AND NOT "2号梯下行命令") OR (NOT "2号梯上行命令" AND NOT "2号梯下行命令")) AND "2号梯电梯停稳信号" AND ("2号梯当前楼层数" = 4) AND "4层外呼上行指示灯";
   IF #_w6 THEN
       "4层外呼上行指示灯" := FALSE;
       "2号梯4层上呼" := FALSE;
       "DB_GC".HallUpCancel[4] := TRUE;
   END_IF;
   #_w7 := (("3层外呼上行指示灯" AND "3层外呼下行指示灯" AND "2号梯上行命令" AND NOT "2号梯下行命令" AND "2号梯本层召唤开门信号") OR (NOT "3层外呼下行指示灯" AND "3层外呼上行指示灯" AND "2号梯本层召唤开门信号" AND "2号梯上行命令" AND NOT "2号梯下行命令") OR (NOT "2号梯上行命令" AND NOT "2号梯下行命令")) AND "2号梯电梯停稳信号" AND ("2号梯当前楼层数" = 3) AND "3层外呼上行指示灯";
   IF #_w7 THEN
       "3层外呼上行指示灯" := FALSE;
       "2号梯3层上呼" := FALSE;
       "DB_GC".HallUpCancel[3] := TRUE;
   END_IF;
   #_w8 := (("2层外呼上行指示灯" AND "2层外呼下行指示灯" AND "2号梯上行命令" AND NOT "2号梯下行命令" AND "2号梯本层召唤开门信号") OR (NOT "2层外呼下行指示灯" AND "2层外呼上行指示灯" AND "2号梯本层召唤开门信号" AND "2号梯上行命令" AND NOT "2号梯下行命令") OR (NOT "2号梯上行命令" AND NOT "2号梯下行命令")) AND "2号梯电梯停稳信号" AND ("2号梯当前楼层数" = 2) AND "2层外呼上行指示灯";
   IF #_w8 THEN
       "2层外呼上行指示灯" := FALSE;
       "2号梯2层上呼" := FALSE;
       "DB_GC".HallUpCancel[2] := TRUE;
   END_IF;
   #_w9 := (("1层外呼上行指示灯" AND "2号梯本层召唤开门信号") OR (NOT "2号梯上行命令" AND NOT "2号梯下行命令")) AND ("2号梯当前楼层数" = 1) AND "1层外呼上行指示灯" AND "2号梯电梯停稳信号";
   IF #_w9 THEN
       "1层外呼上行指示灯" := FALSE;
       "2号梯1层上呼" := FALSE;
       "DB_GC".HallUpCancel[1] := TRUE;
   END_IF;
END_REGION
END_FUNCTION

FUNCTION "2号梯开关门控制" : Void   // FC29, LAD
{ S7_Optimized_Access := 'TRUE' }
VERSION : 0.1
   VAR_TEMP   // added for the SCL form of the ladder/FBD networks
      _w1 : Bool;
   END_VAR
BEGIN

REGION Network 1: 开门使能
